LIN {X 0,Y 362.665,Z 342.074,A -85,B 0,C 180,E1 -13518.879,E2 -13518.879} C_VEL
LIN {X 0,Y 362.673,Z 345.002,A -85,B 0,C 180,E1 -13519.116,E2 -13519.116} C_VEL
LIN {X 0,Y 361.547,Z 357.376,A -85,B 0,C 180,E1 -13520.184,E2 -13520.184} C_VEL
LIN {X 0,Y 360.334,Z 368.054,A -85,B 0,C 180,E1 -13521.361,E2 -13521.361} C_VEL
LIN {X 0,Y 359.164,Z 377.919,A -85,B 0,C 180,E1 -13522.714,E2 -13522.714} C_VEL
LIN {X 0,Y 357.885,Z 387.519,A -85,B 0,C 180,E1 -13524.355,E2 -13524.355} C_VEL
LIN {X 0,Y 356.833,Z 395.168,A -85,B 0,C 180,E1 -13525.991,E2 -13525.991} C_VEL
LIN {X 0,Y 355.858,Z 401.859,A -85,B 0,C 180,E1 -13527.774,E2 -13527.774} C_VEL
LIN {X 0,Y 355.058,Z 407.359,A -85,B 0,C 180,E1 -13529.66,E2 -13529.66} C_VEL
LIN {X 0,Y 354.484,Z 411.392,A -85,B 0,C 180,E1 -13531.512,E2 -13531.512} C_VEL
LIN {X 0,Y 353.919,Z 414.746,A -85,B 0,C 180,E1 -13533.78,E2 -13533.78} C_VEL
LIN {X 0,Y 353.636,Z 416.133,A -85,B 0,C 180,E1 -13535.43,E2 -13535.43} C_VEL
LIN {X 0,Y 353.498,Z 416.697,A -85,B 0,C 180,E1 -13537.32,E2 -13537.32} C_VEL
LIN {X 0,Y 353.475,Z 415.987,A -85,B 0,C 180,E1 -13539.512,E2 -13539.512} C_VEL
LIN {X 0,Y 353.681,Z 413.711,A -85,B 0,C 180,E1 -13541.734,E2 -13541.734} C_VEL
LIN {X 0,Y 353.978,Z 411.14,A -85,B 0,C 180,E1 -13543.308,E2 -13543.308} C_VEL
LIN {X 0,Y 354.296,Z 407.587,A -85,B 0,C 180,E1 -13544.933,E2 -13544.933} C_VEL
LIN {X 0,Y 354.697,Z 403.044,A -85,B 0,C 180,E1 -13546.551,E2 -13546.551} C_VEL
LIN {X 0,Y 355.307,Z 396.31,A -85,B 0,C 180,E1 -13548.437,E2 -13548.437} C_VEL
LIN {X 0,Y 356.124,Z 388.706,A -85,B 0,C 180,E1 -13550.13,E2 -13550.13} C_VEL
LIN {X 0,Y 356.981,Z 379.715,A -85,B 0,C 180,E1 -13551.739,E2 -13551.739} C_VEL
LIN {X 0,Y 357.963,Z 369.677,A -85,B 0,C 180,E1 -13553.19,E2 -13553.19} C_VEL
LIN {X 0,Y 358.986,Z 358.544,A -85,B 0,C 180,E1 -13554.481,E2 -13554.481} C_VEL
LIN {X 0,Y 359.748,Z 347.631,A -85,B 0,C 180,E1 -13555.49,E2 -13555.49} C_VEL
LIN {X 0,Y 360.26,Z 338.398,A -85,B 0,C 180,E1 -13556.184,E2 -13556.184} C_VEL
LIN {X 0,Y 357.076,Z 324.773,A -85,B 0,C 180,E1 -13557.147,E2 -13557.147} C_VEL
LIN {X 0,Y 353.922,Z 312.67,A -85,B 0,C 180,E1 -13557.831,E2 -13557.831} C_VEL
LIN {X 0,Y 353.979,Z 310.393,A -85,B 0,C 180,E1 -13560.24,E2 -13560.24} C_VEL
LIN {X 0,Y 354.41,Z 310.341,A -85,B 0,C 180,E1 -13563.171,E2 -13563.171} C_VEL
LIN {X 0,Y 354.706,Z 310.3,A -85,B 0,C 180,E1 -13566.654,E2 -13566.654} C_VEL
LIN {X 0,Y 354.82,Z 310.289,A -85,B 0,C 180,E1 -13569.113,E2 -13569.113} C_VEL
LIN {X 0,Y 354.881,Z 310.28,A -85,B 0,C 180,E1 -13572.719,E2 -13572.719} C_VEL
LIN {X 0,Y 354.952,Z 310.269,A -85,B 0,C 180,E1 -13576.255,E2 -13576.255} C_VEL
LIN {X 0,Y 354.979,Z 310.265,A -85,B 0,C 180,E1 -13579.736,E2 -13579.736} C_VEL
LIN {X 0,Y 355.101,Z 310.253,A -85,B 0,C 180,E1 -13583.18,E2 -13583.18} C_VEL
LIN {X 0,Y 355.244,Z 310.232,A -85,B 0,C 180,E1 -13587.732,E2 -13587.732} C_VEL
LIN {X 0,Y 355.397,Z 310.213,A -85,B 0,C 180,E1 -13590,E2 -13590} C_VEL
LIN {X 0,Y 355.247,Z 310.234,A -85,B 0,C 180,E1 -13592.268,E2 -13592.268} C_VEL
LIN {X 0,Y 355.1,Z 310.254,A -85,B 0,C 180,E1 -13596.82,E2 -13596.82} C_VEL
LIN {X 0,Y 354.978,Z 310.268,A -85,B 0,C 180,E1 -13600.264,E2 -13600.264} C_VEL
LIN {X 0,Y 354.944,Z 310.271,A -85,B 0,C 180,E1 -13604.019,E2 -13604.019} C_VEL
LIN {X 0,Y 354.923,Z 310.275,A -85,B 0,C 180,E1 -13608.109,E2 -13608.109} C_VEL
LIN {X 0,Y 354.836,Z 310.287,A -85,B 0,C 180,E1 -13612.106,E2 -13612.106} C_VEL
LIN {X 0,Y 354.901,Z 310.277,A -85,B 0,C 180,E1 -13615.828,E2 -13615.828} C_VEL
LIN {X 0,Y 354.855,Z 310.282,A -85,B 0,C 180,E1 -13619.679,E2 -13619.679} C_VEL
LIN {X 0,Y 354.807,Z 310.289,A -85,B 0,C 180,E1 -13623.702,E2 -13623.702} C_VEL
LIN {X 0,Y 354.791,Z 310.289,A -85,B 0,C 180,E1 -13627.248,E2 -13627.248} C_VEL
LIN {X 0,Y 354.789,Z 310.289,A -85,B 0,C 180,E1 -13630.821,E2 -13630.821} C_VEL
LIN {X 0,Y 354.786,Z 310.289,A -85,B 0,C 180,E1 -13632.165,E2 -13632.165} C_VEL
LIN {X 0,Y 354.153,Z 310.373,A -85,B 0,C 180,E1 -13633.111,E2 -13633.111} C_VEL
LIN {X 0,Y 351.293,Z 310.729,A -85,B 0,C 180,E1 -13634.651,E2 -13634.651} C_VEL
LIN {X 0,Y 348.847,Z 311.034,A -85,B 0,C 180,E1 -13635.896,E2 -13635.896} C_VEL
LIN {X 0,Y 347.794,Z 311.16,A -85,B 0,C 180,E1 -13636.861,E2 -13636.861} C_VEL
LIN {X 0,Y 347.709,Z 311.168,A -85,B 0,C 180,E1 -13637.187,E2 -13637.187} C_VEL
LIN {X 0,Y 347.749,Z 311.167,A -85,B 0,C 180,E1 -13640.173,E2 -13640.173} C_VEL
LIN {X 0,Y 347.764,Z 311.163,A -85,B 0,C 180,E1 -13642.68,E2 -13642.68} C_VEL
LIN {X 0,Y 347.75,Z 311.168,A -85,B 0,C 180,E1 -13645.956,E2 -13645.956} C_VEL
LIN {X 0,Y 347.766,Z 311.168,A -85,B 0,C 180,E1 -13649.654,E2 -13649.654} C_VEL
LIN {X 0,Y 347.854,Z 311.153,A -85,B 0,C 180,E1 -13652.745,E2 -13652.745} C_VEL
LIN {X 0,Y 347.788,Z 311.161,A -85,B 0,C 180,E1 -13656.162,E2 -13656.162} C_VEL
LIN {X 0,Y 347.803,Z 311.16,A -85,B 0,C 180,E1 -13659.909,E2 -13659.909} C_VEL
LIN {X 0,Y 347.836,Z 311.157,A -85,B 0,C 180,E1 -13663.569,E2 -13663.569} C_VEL
LIN {X 0,Y 347.894,Z 311.152,A -85,B 0,C 180,E1 -13667.161,E2 -13667.161} C_VEL
LIN {X 0,Y 347.939,Z 311.144,A -85,B 0,C 180,E1 -13670.701,E2 -13670.701} C_VEL
LIN {X 0,Y 348.086,Z 311.129,A -85,B 0,C 180,E1 -13673.042,E2 -13673.042} C_VEL
LIN {X 0,Y 348.207,Z 311.108,A -85,B 0,C 180,E1 -13677.687,E2 -13677.687} C_VEL
LIN {X 0,Y 348.328,Z 311.093,A -85,B 0,C 180,E1 -13680,E2 -13680} C_VEL
LIN {X 0,Y 348.199,Z 311.11,A -85,B 0,C 180,E1 -13682.314,E2 -13682.314} C_VEL
LIN {X 0,Y 348.072,Z 311.129,A -85,B 0,C 180,E1 -13686.958,E2 -13686.958} C_VEL
LIN {X 0,Y 347.901,Z 311.15,A -85,B 0,C 180,E1 -13690.475,E2 -13690.475} C_VEL
LIN {X 0,Y 347.902,Z 311.148,A -85,B 0,C 180,E1 -13694.15,E2 -13694.15} C_VEL
LIN {X 0,Y 347.832,Z 311.158,A -85,B 0,C 180,E1 -13698.259,E2 -13698.259} C_VEL
LIN {X 0,Y 347.771,Z 311.163,A -85,B 0,C 180,E1 -13701.626,E2 -13701.626} C_VEL
LIN {X 0,Y 347.796,Z 311.16,A -85,B 0,C 180,E1 -13705.11,E2 -13705.11} C_VEL
LIN {X 0,Y 347.76,Z 311.164,A -85,B 0,C 180,E1 -13709.014,E2 -13709.014} C_VEL
LIN {X 0,Y 347.745,Z 311.166,A -85,B 0,C 180,E1 -13713.071,E2 -13713.071} C_VEL
LIN {X 0,Y 347.773,Z 311.167,A -85,B 0,C 180,E1 -13716.065,E2 -13716.065} C_VEL
LIN {X 0,Y 347.755,Z 311.165,A -85,B 0,C 180,E1 -13718.793,E2 -13718.793} C_VEL
LIN {X 0,Y 347.753,Z 311.169,A -85,B 0,C 180,E1 -13721.83,E2 -13721.83} C_VEL
LIN {X 0,Y 347.791,Z 311.271,A -85,B 0,C 180,E1 -13724.819,E2 -13724.819} C_VEL
LIN {X 0,Y 348.908,Z 317.424,A -85,B 0,C 180,E1 -13728.339,E2 -13728.339} C_VEL
LIN {X 0,Y 349.989,Z 323.328,A -85,B 0,C 180,E1 -13731.55,E2 -13731.55} C_VEL
LIN {X 0,Y 350.336,Z 327.895,A -85,B 0,C 180,E1 -13733.897,E2 -13733.897} C_VEL
LIN {X 0,Y 349.502,Z 334.535,A -85,B 0,C 180,E1 -13737.116,E2 -13737.116} C_VEL
LIN {X 0,Y 348.554,Z 342.889,A -85,B 0,C 180,E1 -13741.058,E2 -13741.058} C_VEL
LIN {X 0,Y 347.745,Z 351.233,A -85,B 0,C 180,E1 -13744.886,E2 -13744.886} C_VEL
LIN {X 0,Y 347.106,Z 359.56,A -85,B 0,C 180,E1 -13748.652,E2 -13748.652} C_VEL
LIN {X 0,Y 346.983,Z 362.085,A -85,B 0,C 180,E1 -13749.782,E2 -13749.782} C_VEL
LIN {X 0,Y 348.977,Z 376.53,A -85,B 0,C 180,E1 -13750.44,E2 -13750.44} C_VEL
LIN {X 0,Y 350.363,Z 388.913,A -85,B 0,C 180,E1 -13751.22,E2 -13751.22} C_VEL
LIN {X 0,Y 351.311,Z 401.597,A -85,B 0,C 180,E1 -13752.237,E2 -13752.237} C_VEL
LIN {X 0,Y 351.019,Z 407.958,A -85,B 0,C 180,E1 -13752.823,E2 -13752.823} C_VEL
LIN {X 0,Y 349.791,Z 419.655,A -85,B 0,C 180,E1 -13754.112,E2 -13754.112} C_VEL
LIN {X 0,Y 348.824,Z 429.132,A -85,B 0,C 180,E1 -13755.41,E2 -13755.41} C_VEL
LIN {X 0,Y 348.012,Z 437.864,A -85,B 0,C 180,E1 -13756.868,E2 -13756.868} C_VEL
LIN {X 0,Y 347.235,Z 446.325,A -85,B 0,C 180,E1 -13758.619,E2 -13758.619} C_VEL
LIN {X 0,Y 346.77,Z 453.136,A -85,B 0,C 180,E1 -13760.375,E2 -13760.375} C_VEL
LIN {X 0,Y 346.461,Z 459.371,A -85,B 0,C 180,E1 -13762.423,E2 -13762.423} C_VEL
LIN {X 0,Y 346.36,Z 463.393,A -85,B 0,C 180,E1 -13764.177,E2 -13764.177} C_VEL
LIN {X 0,Y 346.372,Z 465.449,A -85,B 0,C 180,E1 -13765.345,E2 -13765.345} C_VEL
LIN {X 0,Y 346.529,Z 468.273,A -85,B 0,C 180,E1 -13767.675,E2 -13767.675} C_VEL
LIN {X 0,Y 346.531,Z 469.026,A -85,B 0,C 180,E1 -13768.838,E2 -13768.838} C_VEL
LIN {X 0,Y 346.546,Z 469.344,A -85,B 0,C 180,E1 -13770,E2 -13770} C_VEL
LIN {X 0,Y 346.51,Z 469.256,A -85,B 0,C 180,E1 -13771.162,E2 -13771.162} C_VEL
LIN {X 0,Y 346.497,Z 468.769,A -85,B 0,C 180,E1 -13772.325,E2 -13772.325} C_VEL
LIN {X 0,Y 346.337,Z 467.838,A -85,B 0,C 180,E1 -13773.49,E2 -13773.49} C_VEL
LIN {X 0,Y 346.321,Z 466.48,A -85,B 0,C 180,E1 -13774.656,E2 -13774.656} C_VEL
LIN {X 0,Y 346.243,Z 464.483,A -85,B 0,C 180,E1 -13775.956,E2 -13775.956} C_VEL
LIN {X 0,Y 346.409,Z 461.197,A -85,B 0,C 180,E1 -13777.578,E2 -13777.578} C_VEL
LIN {X 0,Y 346.684,Z 456.619,A -85,B 0,C 180,E1 -13779.333,E2 -13779.333} C_VEL
LIN {X 0,Y 347.291,Z 449.778,A -85,B 0,C 180,E1 -13781.38,E2 -13781.38} C_VEL
LIN {X 0,Y 348.248,Z 442.357,A -85,B 0,C 180,E1 -13783.123,E2 -13783.123} C_VEL
LIN {X 0,Y 349.358,Z 433.079,A -85,B 0,C 180,E1 -13784.888,E2 -13784.888} C_VEL
LIN {X 0,Y 350.468,Z 423.926,A -85,B 0,C 180,E1 -13786.305,E2 -13786.305} C_VEL
LIN {X 0,Y 352.052,Z 412.428,A -85,B 0,C 180,E1 -13787.724,E2 -13787.724} C_VEL
LIN {X 0,Y 352.831,Z 404.137,A -85,B 0,C 180,E1 -13788.585,E2 -13788.585} C_VEL
LIN {X 0,Y 352.469,Z 391.587,A -85,B 0,C 180,E1 -13789.73,E2 -13789.73} C_VEL
LIN {X 0,Y 351.594,Z 381.993,A -85,B 0,C 180,E1 -13790.475,E2 -13790.475} C_VEL
LIN {X 0,Y 349.591,Z 369.477,A -85,B 0,C 180,E1 -13791.313,E2 -13791.313} C_VEL
LIN {X 0,Y 347.227,Z 358.557,A -85,B 0,C 180,E1 -13791.943,E2 -13791.943} C_VEL
LIN {X 0,Y 347.858,Z 350.269,A -85,B 0,C 180,E1 -13795.746,E2 -13795.746} C_VEL
LIN {X 0,Y 348.678,Z 342.519,A -85,B 0,C 180,E1 -13799.442,E2 -13799.442} C_VEL
LIN {X 0,Y 349.811,Z 334.351,A -85,B 0,C 180,E1 -13803.539,E2 -13803.539} C_VEL
LIN {X 0,Y 350.574,Z 329.466,A -85,B 0,C 180,E1 -13806.13,E2 -13806.13} C_VEL
LIN {X 0,Y 350.555,Z 326.753,A -85,B 0,C 180,E1 -13807.696,E2 -13807.696} C_VEL
LIN {X 0,Y 349.769,Z 321.77,A -85,B 0,C 180,E1 -13810.835,E2 -13810.835} C_VEL
LIN {X 0,Y 349.048,Z 317.863,A -85,B 0,C 180,E1 -13813.543,E2 -13813.543} C_VEL
LIN {X 0,Y 348.264,Z 313.827,A -85,B 0,C 180,E1 -13816.676,E2 -13816.676} C_VEL
LIN {X 0,Y 347.745,Z 311.176,A -85,B 0,C 180,E1 -13819.035,E2 -13819.035} C_VEL
LIN {X 0,Y 347.769,Z 311.169,A -85,B 0,C 180,E1 -13822.68,E2 -13822.68} C_VEL
LIN {X 0,Y 347.752,Z 311.169,A -85,B 0,C 180,E1 -13825.956,E2 -13825.956} C_VEL
LIN {X 0,Y 347.768,Z 311.167,A -85,B 0,C 180,E1 -13829.654,E2 -13829.654} C_VEL
LIN {X 0,Y 347.856,Z 311.156,A -85,B 0,C 180,E1 -13832.745,E2 -13832.745} C_VEL
LIN {X 0,Y 347.793,Z 311.162,A -85,B 0,C 180,E1 -13836.162,E2 -13836.162} C_VEL
LIN {X 0,Y 347.822,Z 311.157,A -85,B 0,C 180,E1 -13839.91,E2 -13839.91} C_VEL
LIN {X 0,Y 347.871,Z 311.151,A -85,B 0,C 180,E1 -13842.359,E2 -13842.359} C_VEL
LIN {X 0,Y 347.901,Z 311.15,A -85,B 0,C 180,E1 -13845.971,E2 -13845.971} C_VEL
LIN {X 0,Y 347.901,Z 311.149,A -85,B 0,C 180,E1 -13849.525,E2 -13849.525} C_VEL
LIN {X 0,Y 348.072,Z 311.127,A -85,B 0,C 180,E1 -13853.042,E2 -13853.042} C_VEL
LIN {X 0,Y 348.21,Z 311.111,A -85,B 0,C 180,E1 -13857.686,E2 -13857.686} C_VEL
LIN {X 0,Y 348.35,Z 311.096,A -85,B 0,C 180,E1 -13860,E2 -13860} C_VEL
LIN {X 0,Y 348.213,Z 311.111,A -85,B 0,C 180,E1 -13862.313,E2 -13862.313} C_VEL
LIN {X 0,Y 348.069,Z 311.13,A -85,B 0,C 180,E1 -13866.958,E2 -13866.958} C_VEL
LIN {X 0,Y 347.992,Z 311.14,A -85,B 0,C 180,E1 -13868.268,E2 -13868.268} C_VEL
LIN {X 0,Y 347.82,Z 313.428,A -85,B 0,C 180,E1 -13871.657,E2 -13871.657} C_VEL
LIN {X 0,Y 347.641,Z 316.115,A -85,B 0,C 180,E1 -13875.237,E2 -13875.237} C_VEL
LIN {X 0,Y 347.621,Z 317.069,A -85,B 0,C 180,E1 -13876.253,E2 -13876.253} C_VEL
LIN {X 0,Y 352.283,Z 329.9,A -85,B 0,C 180,E1 -13877.263,E2 -13877.263} C_VEL
LIN {X 0,Y 355.595,Z 341.553,A -85,B 0,C 180,E1 -13878.3,E2 -13878.3} C_VEL
LIN {X 0,Y 356.194,Z 344.142,A -85,B 0,C 180,E1 -13878.551,E2 -13878.551} C_VEL
LIN {X 0,Y 355.247,Z 355.316,A -85,B 0,C 180,E1 -13879.502,E2 -13879.502} C_VEL
LIN {X 0,Y 354.027,Z 365.973,A -85,B 0,C 180,E1 -13880.632,E2 -13880.632} C_VEL
LIN {X 0,Y 352.857,Z 375.772,A -85,B 0,C 180,E1 -13881.929,E2 -13881.929} C_VEL
LIN {X 0,Y 351.41,Z 385.788,A -85,B 0,C 180,E1 -13883.577,E2 -13883.577} C_VEL
LIN {X 0,Y 350.332,Z 393.517,A -85,B 0,C 180,E1 -13885.156,E2 -13885.156} C_VEL
LIN {X 0,Y 349.251,Z 400.486,A -85,B 0,C 180,E1 -13886.918,E2 -13886.918} C_VEL
LIN {X 0,Y 348.303,Z 406.735,A -85,B 0,C 180,E1 -13888.964,E2 -13888.964} C_VEL
LIN {X 0,Y 347.584,Z 411.468,A -85,B 0,C 180,E1 -13891.037,E2 -13891.037} C_VEL
LIN {X 0,Y 346.981,Z 414.757,A -85,B 0,C 180,E1 -13893.153,E2 -13893.153} C_VEL
LIN {X 0,Y 346.698,Z 416.206,A -85,B 0,C 180,E1 -13894.583,E2 -13894.583} C_VEL
LIN {X 0,Y 346.501,Z 417.022,A -85,B 0,C 180,E1 -13896.029,E2 -13896.029} C_VEL
LIN {X 0,Y 346.402,Z 417.224,A -85,B 0,C 180,E1 -13897.696,E2 -13897.696} C_VEL
LIN {X 0,Y 346.395,Z 416.473,A -85,B 0,C 180,E1 -13899.557,E2 -13899.557} C_VEL
LIN {X 0,Y 346.554,Z 414.734,A -85,B 0,C 180,E1 -13901.379,E2 -13901.379} C_VEL
LIN {X 0,Y 346.943,Z 411.334,A -85,B 0,C 180,E1 -13903.53,E2 -13903.53} C_VEL
LIN {X 0,Y 347.269,Z 407.89,A -85,B 0,C 180,E1 -13905.099,E2 -13905.099} C_VEL
LIN {X 0,Y 347.789,Z 402.248,A -85,B 0,C 180,E1 -13907.075,E2 -13907.075} C_VEL
LIN {X 0,Y 348.349,Z 396.36,A -85,B 0,C 180,E1 -13908.702,E2 -13908.702} C_VEL
LIN {X 0,Y 349.146,Z 389.139,A -85,B 0,C 180,E1 -13910.326,E2 -13910.326} C_VEL
LIN {X 0,Y 350.002,Z 380.39,A -85,B 0,C 180,E1 -13911.923,E2 -13911.923} C_VEL
LIN {X 0,Y 350.969,Z 370.922,A -85,B 0,C 180,E1 -13913.329,E2 -13913.329} C_VEL
LIN {X 0,Y 351.978,Z 360.255,A -85,B 0,C 180,E1 -13914.616,E2 -13914.616} C_VEL
LIN {X 0,Y 352.791,Z 349.433,A -85,B 0,C 180,E1 -13915.666,E2 -13915.666} C_VEL
LIN {X 0,Y 353.507,Z 340.69,A -85,B 0,C 180,E1 -13916.346,E2 -13916.346} C_VEL
LIN {X 0,Y 350.753,Z 328.113,A -85,B 0,C 180,E1 -13917.291,E2 -13917.291} C_VEL
LIN {X 0,Y 347.373,Z 315.098,A -85,B 0,C 180,E1 -13918.049,E2 -13918.049} C_VEL
LIN {X 0,Y 346.908,Z 313.147,A -85,B 0,C 180,E1 -13918.172,E2 -13918.172} C_VEL
LIN {X 0,Y 346.898,Z 311.778,A -85,B 0,C 180,E1 -13919.569,E2 -13919.569} C_VEL
LIN {X 0,Y 347.058,Z 311.255,A -85,B 0,C 180,E1 -13920.921,E2 -13920.921} C_VEL
LIN {X 0,Y 347.381,Z 311.215,A -85,B 0,C 180,E1 -13923.571,E2 -13923.571} C_VEL
LIN {X 0,Y 347.632,Z 311.18,A -85,B 0,C 180,E1 -13926.15,E2 -13926.15} C_VEL
LIN {X 0,Y 347.796,Z 311.16,A -85,B 0,C 180,E1 -13929.908,E2 -13929.908} C_VEL
LIN {X 0,Y 347.833,Z 311.156,A -85,B 0,C 180,E1 -13933.568,E2 -13933.568} C_VEL
LIN {X 0,Y 347.891,Z 311.152,A -85,B 0,C 180,E1 -13937.16,E2 -13937.16} C_VEL
LIN {X 0,Y 347.942,Z 311.145,A -85,B 0,C 180,E1 -13940.701,E2 -13940.701} C_VEL
LIN {X 0,Y 348.051,Z 311.128,A -85,B 0,C 180,E1 -13944.205,E2 -13944.205} C_VEL
LIN {X 0,Y 348.207,Z 311.108,A -85,B 0,C 180,E1 -13947.686,E2 -13947.686} C_VEL
LIN {X 0,Y 348.346,Z 311.091,A -85,B 0,C 180,E1 -13950,E2 -13950} C_VEL
LIN {X 0,Y 348.209,Z 311.11,A -85,B 0,C 180,E1 -13952.313,E2 -13952.313} C_VEL
LIN {X 0,Y 348.068,Z 311.128,A -85,B 0,C 180,E1 -13956.958,E2 -13956.958} C_VEL
LIN {X 0,Y 347.929,Z 311.148,A -85,B 0,C 180,E1 -13960.474,E2 -13960.474} C_VEL
LIN {X 0,Y 347.899,Z 311.15,A -85,B 0,C 180,E1 -13964.15,E2 -13964.15} C_VEL
LIN {X 0,Y 347.892,Z 311.153,A -85,B 0,C 180,E1 -13968.29,E2 -13968.29} C_VEL
LIN {X 0,Y 347.79,Z 311.161,A -85,B 0,C 180,E1 -13971.635,E2 -13971.635} C_VEL
LIN {X 0,Y 347.813,Z 311.157,A -85,B 0,C 180,E1 -13975.109,E2 -13975.109} C_VEL
LIN {X 0,Y 347.812,Z 311.159,A -85,B 0,C 180,E1 -13977.694,E2 -13977.694} C_VEL
LIN {X 0,Y 347.765,Z 311.167,A -85,B 0,C 180,E1 -13980.347,E2 -13980.347} C_VEL
LIN {X 0,Y 347.745,Z 311.168,A -85,B 0,C 180,E1 -13984.464,E2 -13984.464} C_VEL
LIN {X 0,Y 347.775,Z 311.167,A -85,B 0,C 180,E1 -13987.989,E2 -13987.989} C_VEL
LIN {X 0,Y 347.752,Z 311.17,A -85,B 0,C 180,E1 -13991.83,E2 -13991.83} C_VEL
LIN {X 0,Y 347.707,Z 311.171,A -85,B 0,C 180,E1 -13995.027,E2 -13995.027} C_VEL
LIN {X 0,Y 347.709,Z 311.168,A -85,B 0,C 180,E1 -13997.187,E2 -13997.187} C_VEL
LIN {X 0,Y 347.053,Z 311.255,A -85,B 0,C 180,E1 -13998.154,E2 -13998.154} C_VEL
LIN {X 0,Y 344.233,Z 311.608,A -85,B 0,C 180,E1 -13999.728,E2 -13999.728} C_VEL
LIN {X 0,Y 341.834,Z 311.907,A -85,B 0,C 180,E1 -14001.001,E2 -14001.001} C_VEL
LIN {X 0,Y 340.79,Z 312.035,A -85,B 0,C 180,E1 -14001.986,E2 -14001.986} C_VEL
LIN {X 0,Y 340.698,Z 312.044,A -85,B 0,C 180,E1 -14002.32,E2 -14002.32} C_VEL
LIN {X 0,Y 340.725,Z 312.046,A -85,B 0,C 180,E1 -14005.596,E2 -14005.596} C_VEL
LIN {X 0,Y 340.706,Z 312.044,A -85,B 0,C 180,E1 -14008.956,E2 -14008.956} C_VEL
LIN {X 0,Y 340.781,Z 312.033,A -85,B 0,C 180,E1 -14012.474,E2 -14012.474} C_VEL
LIN {X 0,Y 340.757,Z 312.04,A -85,B 0,C 180,E1 -14015.639,E2 -14015.639} C_VEL
LIN {X 0,Y 340.733,Z 312.043,A -85,B 0,C 180,E1 -14019.473,E2 -14019.473} C_VEL
LIN {X 0,Y 340.795,Z 312.032,A -85,B 0,C 180,E1 -14021.981,E2 -14021.981} C_VEL
LIN {X 0,Y 340.873,Z 312.023,A -85,B 0,C 180,E1 -14025.705,E2 -14025.705} C_VEL
LIN {X 0,Y 340.852,Z 312.028,A -85,B 0,C 180,E1 -14029.306,E2 -14029.306} C_VEL
LIN {X 0,Y 341.053,Z 312.004,A -85,B 0,C 180,E1 -14032.898,E2 -14032.898} C_VEL
LIN {X 0,Y 341.169,Z 311.985,A -85,B 0,C 180,E1 -14037.639,E2 -14037.639} C_VEL
LIN {X 0,Y 341.279,Z 311.971,A -85,B 0,C 180,E1 -14040,E2 -14040} C_VEL
LIN {X 0,Y 341.16,Z 311.987,A -85,B 0,C 180,E1 -14042.361,E2 -14042.361} C_VEL
LIN {X 0,Y 341.02,Z 312.006,A -85,B 0,C 180,E1 -14047.103,E2 -14047.103} C_VEL
LIN {X 0,Y 340.853,Z 312.029,A -85,B 0,C 180,E1 -14050.695,E2 -14050.695} C_VEL
LIN {X 0,Y 340.867,Z 312.026,A -85,B 0,C 180,E1 -14054.325,E2 -14054.325} C_VEL
LIN {X 0,Y 340.789,Z 312.037,A -85,B 0,C 180,E1 -14058.44,E2 -14058.44} C_VEL
LIN {X 0,Y 340.721,Z 312.041,A -85,B 0,C 180,E1 -14061.842,E2 -14061.842} C_VEL
LIN {X 0,Y 340.748,Z 312.038,A -85,B 0,C 180,E1 -14065.667,E2 -14065.667} C_VEL
LIN {X 0,Y 340.735,Z 312.04,A -85,B 0,C 180,E1 -14069.672,E2 -14069.672} C_VEL
LIN {X 0,Y 340.697,Z 312.046,A -85,B 0,C 180,E1 -14073.846,E2 -14073.846} C_VEL
LIN {X 0,Y 340.708,Z 312.043,A -85,B 0,C 180,E1 -14076.742,E2 -14076.742} C_VEL
LIN {X 0,Y 340.691,Z 312.049,A -85,B 0,C 180,E1 -14080.247,E2 -14080.247} C_VEL
LIN {X 0,Y 340.676,Z 312.05,A -85,B 0,C 180,E1 -14083.777,E2 -14083.777} C_VEL
LIN {X 0,Y 340.745,Z 312.183,A -85,B 0,C 180,E1 -14084.529,E2 -14084.529} C_VEL
LIN {X 0,Y 341.943,Z 318.683,A -85,B 0,C 180,E1 -14088.333,E2 -14088.333} C_VEL
LIN {X 0,Y 343.148,Z 325.501,A -85,B 0,C 180,E1 -14092.089,E2 -14092.089} C_VEL
LIN {X 0,Y 343.319,Z 328.345,A -85,B 0,C 180,E1 -14093.583,E2 -14093.583} C_VEL
LIN {X 0,Y 342.676,Z 333.956,A -85,B 0,C 180,E1 -14096.375,E2 -14096.375} C_VEL
LIN {X 0,Y 341.648,Z 342.287,A -85,B 0,C 180,E1 -14100.416,E2 -14100.416} C_VEL
LIN {X 0,Y 340.757,Z 350.593,A -85,B 0,C 180,E1 -14104.334,E2 -14104.334} C_VEL
LIN {X 0,Y 340.066,Z 359.448,A -85,B 0,C 180,E1 -14108.435,E2 -14108.435} C_VEL
LIN {X 0,Y 339.928,Z 361.604,A -85,B 0,C 180,E1 -14109.422,E2 -14109.422} C_VEL
LIN {X 0,Y 341.965,Z 376.241,A -85,B 0,C 180,E1 -14110.111,E2 -14110.111} C_VEL
LIN {X 0,Y 343.395,Z 389.241,A -85,B 0,C 180,E1 -14110.958,E2 -14110.958} C_VEL
LIN {X 0,Y 344.251,Z 400.211,A -85,B 0,C 180,E1 -14111.86,E2 -14111.86} C_VEL
LIN {X 0,Y 344.242,Z 406.734,A -85,B 0,C 180,E1 -14112.474,E2 -14112.474} C_VEL
LIN {X 0,Y 343.04,Z 417.408,A -85,B 0,C 180,E1 -14113.638,E2 -14113.638} C_VEL
LIN {X 0,Y 342.012,Z 427.255,A -85,B 0,C 180,E1 -14114.974,E2 -14114.974} C_VEL
LIN {X 0,Y 341.265,Z 435.32,A -85,B 0,C 180,E1 -14116.3,E2 -14116.3} C_VEL
LIN {X 0,Y 340.41,Z 444.216,A -85,B 0,C 180,E1 -14118.085,E2 -14118.085} C_VEL
LIN {X 0,Y 339.777,Z 451.344,A -85,B 0,C 180,E1 -14119.874,E2 -14119.874} C_VEL
LIN {X 0,Y 339.453,Z 457.025,A -85,B 0,C 180,E1 -14121.667,E2 -14121.667} C_VEL
LIN {X 0,Y 339.338,Z 462.166,A -85,B 0,C 180,E1 -14123.788,E2 -14123.788} C_VEL
LIN {X 0,Y 339.305,Z 464.811,A -85,B 0,C 180,E1 -14125.247,E2 -14125.247} C_VEL
LIN {X 0,Y 339.28,Z 466.443,A -85,B 0,C 180,E1 -14126.437,E2 -14126.437} C_VEL
LIN {X 0,Y 339.462,Z 467.672,A -85,B 0,C 180,E1 -14127.627,E2 -14127.627} C_VEL
LIN {X 0,Y 339.465,Z 468.458,A -85,B 0,C 180,E1 -14128.814,E2 -14128.814} C_VEL
LIN {X 0,Y 339.476,Z 468.792,A -85,B 0,C 180,E1 -14130,E2 -14130} C_VEL
LIN {X 0,Y 339.445,Z 468.719,A -85,B 0,C 180,E1 -14131.186,E2 -14131.186} C_VEL
LIN {X 0,Y 339.413,Z 468.246,A -85,B 0,C 180,E1 -14132.373,E2 -14132.373} C_VEL
LIN {X 0,Y 339.251,Z 467.349,A -85,B 0,C 180,E1 -14133.563,E2 -14133.563} C_VEL
LIN {X 0,Y 339.226,Z 466.01,A -85,B 0,C 180,E1 -14134.754,E2 -14134.754} C_VEL
LIN {X 0,Y 339.227,Z 463.224,A -85,B 0,C 180,E1 -14136.543,E2 -14136.543} C_VEL
LIN {X 0,Y 339.419,Z 459.417,A -85,B 0,C 180,E1 -14138.334,E2 -14138.334} C_VEL
LIN {X 0,Y 339.781,Z 454.495,A -85,B 0,C 180,E1 -14140.126,E2 -14140.126} C_VEL
LIN {X 0,Y 340.621,Z 447.176,A -85,B 0,C 180,E1 -14142.21,E2 -14142.21} C_VEL
LIN {X 0,Y 341.584,Z 439.32,A -85,B 0,C 180,E1 -14143.99,E2 -14143.99} C_VEL
LIN {X 0,Y 342.628,Z 431.371,A -85,B 0,C 180,E1 -14145.466,E2 -14145.466} C_VEL
LIN {X 0,Y 344.099,Z 420.723,A -85,B 0,C 180,E1 -14147.074,E2 -14147.074} C_VEL
LIN {X 0,Y 345.625,Z 410.03,A -85,B 0,C 180,E1 -14148.372,E2 -14148.372} C_VEL
LIN {X 0,Y 346.063,Z 403.049,A -85,B 0,C 180,E1 -14149.105,E2 -14149.105} C_VEL
LIN {X 0,Y 345.732,Z 391.118,A -85,B 0,C 180,E1 -14150.217,E2 -14150.217} C_VEL
LIN {X 0,Y 344.502,Z 379.491,A -85,B 0,C 180,E1 -14151.143,E2 -14151.143} C_VEL
LIN {X 0,Y 342.3,Z 366.872,A -85,B 0,C 180,E1 -14152.007,E2 -14152.007} C_VEL
LIN {X 0,Y 340.246,Z 357.904,A -85,B 0,C 180,E1 -14152.553,E2 -14152.553} C_VEL
LIN {X 0,Y 340.918,Z 349.948,A -85,B 0,C 180,E1 -14156.31,E2 -14156.31} C_VEL
LIN {X 0,Y 341.66,Z 343.272,A -85,B 0,C 180,E1 -14159.583,E2 -14159.583} C_VEL
LIN {X 0,Y 342.817,Z 335.455,A -85,B 0,C 180,E1 -14163.609,E2 -14163.609} C_VEL
LIN {X 0,Y 343.614,Z 330.352,A -85,B 0,C 180,E1 -14166.381,E2 -14166.381} C_VEL
LIN {X 0,Y 343.574,Z 327.877,A -85,B 0,C 180,E1 -14167.856,E2 -14167.856} C_VEL
LIN {X 0,Y 342.794,Z 323.002,A -85,B 0,C 180,E1 -14171.001,E2 -14171.001} C_VEL
LIN {X 0,Y 341.911,Z 318.413,A -85,B 0,C 180,E1 -14174.337,E2 -14174.337} C_VEL
LIN {X 0,Y 341.101,Z 314.11,A -85,B 0,C 180,E1 -14177.88,E2 -14177.88} C_VEL
LIN {X 0,Y 340.723,Z 312.047,A -85,B 0,C 180,E1 -14180,E2 -14180} C_VEL
LIN {X 0,Y 340.715,Z 312.044,A -85,B 0,C 180,E1 -14183.559,E2 -14183.559} C_VEL
LIN {X 0,Y 340.698,Z 312.049,A -85,B 0,C 180,E1 -14186.154,E2 -14186.154} C_VEL
LIN {X 0,Y 340.778,Z 312.038,A -85,B 0,C 180,E1 -14190.333,E2 -14190.333} C_VEL
LIN {X 0,Y 340.809,Z 312.033,A -85,B 0,C 180,E1 -14193.02,E2 -14193.02} C_VEL
LIN {X 0,Y 340.733,Z 312.043,A -85,B 0,C 180,E1 -14196.927,E2 -14196.927} C_VEL
LIN {X 0,Y 340.799,Z 312.035,A -85,B 0,C 180,E1 -14200.734,E2 -14200.734} C_VEL
LIN {X 0,Y 340.791,Z 312.037,A -85,B 0,C 180,E1 -14203.219,E2 -14203.219} C_VEL
LIN {X 0,Y 340.849,Z 312.025,A -85,B 0,C 180,E1 -14206.89,E2 -14206.89} C_VEL
LIN {X 0,Y 340.886,Z 312.024,A -85,B 0,C 180,E1 -14210.506,E2 -14210.506} C_VEL
LIN {X 0,Y 341.029,Z 312.006,A -85,B 0,C 180,E1 -14214.086,E2 -14214.086} C_VEL
LIN {X 0,Y 341.172,Z 311.987,A -85,B 0,C 180,E1 -14217.639,E2 -14217.639} C_VEL
LIN {X 0,Y 341.3,Z 311.974,A -85,B 0,C 180,E1 -14220,E2 -14220} C_VEL
LIN {X 0,Y 341.174,Z 311.988,A -85,B 0,C 180,E1 -14222.361,E2 -14222.361} C_VEL
LIN {X 0,Y 341.015,Z 312.009,A -85,B 0,C 180,E1 -14227.103,E2 -14227.103} C_VEL
LIN {X 0,Y 340.967,Z 312.304,A -85,B 0,C 180,E1 -14228.356,E2 -14228.356} C_VEL
LIN {X 0,Y 340.806,Z 314.786,A -85,B 0,C 180,E1 -14231.901,E2 -14231.901} C_VEL
LIN {X 0,Y 340.621,Z 317.483,A -85,B 0,C 180,E1 -14235.559,E2 -14235.559} C_VEL
LIN {X 0,Y 340.601,Z 317.545,A -85,B 0,C 180,E1 -14235.636,E2 -14235.636} C_VEL
LIN {X 0,Y 342.771,Z 323.304,A -85,B 0,C 180,E1 -14236.091,E2 -14236.091} C_VEL
LIN {X 0,Y 346.749,Z 334.691,A -85,B 0,C 180,E1 -14237.091,E2 -14237.091} C_VEL
LIN {X 0,Y 349.601,Z 345.658,A -85,B 0,C 180,E1 -14238.155,E2 -14238.155} C_VEL
LIN {X 0,Y 348.537,Z 357.633,A -85,B 0,C 180,E1 -14239.221,E2 -14239.221} C_VEL
LIN {X 0,Y 347.262,Z 368.127,A -85,B 0,C 180,E1 -14240.397,E2 -14240.397} C_VEL
LIN {X 0,Y 345.826,Z 378.965,A -85,B 0,C 180,E1 -14241.927,E2 -14241.927} C_VEL
LIN {X 0,Y 344.561,Z 387.33,A -85,B 0,C 180,E1 -14243.383,E2 -14243.383} C_VEL
LIN {X 0,Y 343.308,Z 395.452,A -85,B 0,C 180,E1 -14245.137,E2 -14245.137} C_VEL
LIN {X 0,Y 342.26,Z 401.842,A -85,B 0,C 180,E1 -14246.856,E2 -14246.856} C_VEL
LIN {X 0,Y 341.266,Z 407.929,A -85,B 0,C 180,E1 -14248.944,E2 -14248.944} C_VEL
LIN {X 0,Y 340.524,Z 412.465,A -85,B 0,C 180,E1 -14251.062,E2 -14251.062} C_VEL
LIN {X 0,Y 340.082,Z 414.717,A -85,B 0,C 180,E1 -14252.5,E2 -14252.5} C_VEL
LIN {X 0,Y 339.706,Z 416.519,A -85,B 0,C 180,E1 -14254.153,E2 -14254.153} C_VEL
LIN {X 0,Y 339.435,Z 417.654,A -85,B 0,C 180,E1 -14256.147,E2 -14256.147} C_VEL
LIN {X 0,Y 339.31,Z 417.594,A -85,B 0,C 180,E1 -14258.417,E2 -14258.417} C_VEL
LIN {X 0,Y 339.357,Z 416.669,A -85,B 0,C 180,E1 -14259.98,E2 -14259.98} C_VEL
LIN {X 0,Y 339.54,Z 414.687,A -85,B 0,C 180,E1 -14261.828,E2 -14261.828} C_VEL
LIN {X 0,Y 339.892,Z 411.741,A -85,B 0,C 180,E1 -14263.639,E2 -14263.639} C_VEL
LIN {X 0,Y 340.344,Z 406.901,A -85,B 0,C 180,E1 -14265.78,E2 -14265.78} C_VEL
LIN {X 0,Y 340.845,Z 401.927,A -85,B 0,C 180,E1 -14267.455,E2 -14267.455} C_VEL
LIN {X 0,Y 341.466,Z 395.79,A -85,B 0,C 180,E1 -14269.124,E2 -14269.124} C_VEL
LIN {X 0,Y 342.34,Z 387.757,A -85,B 0,C 180,E1 -14270.885,E2 -14270.885} C_VEL
LIN {X 0,Y 343.346,Z 378.445,A -85,B 0,C 180,E1 -14272.537,E2 -14272.537} C_VEL
LIN {X 0,Y 344.367,Z 368.637,A -85,B 0,C 180,E1 -14273.941,E2 -14273.941} C_VEL
LIN {X 0,Y 345.379,Z 357.121,A -85,B 0,C 180,E1 -14275.266,E2 -14275.266} C_VEL
LIN {X 0,Y 346.346,Z 345.74,A -85,B 0,C 180,E1 -14276.301,E2 -14276.301} C_VEL
LIN {X 0,Y 346.537,Z 340.847,A -85,B 0,C 180,E1 -14276.68,E2 -14276.68} C_VEL
LIN {X 0,Y 343.596,Z 328.031,A -85,B 0,C 180,E1 -14277.655,E2 -14277.655} C_VEL
LIN {X 0,Y 340.145,Z 315.11,A -85,B 0,C 180,E1 -14278.423,E2 -14278.423} C_VEL
LIN {X 0,Y 339.838,Z 313.637,A -85,B 0,C 180,E1 -14278.517,E2 -14278.517} C_VEL
LIN {X 0,Y 339.905,Z 312.145,A -85,B 0,C 180,E1 -14280.274,E2 -14280.274} C_VEL
LIN {X 0,Y 340.293,Z 312.097,A -85,B 0,C 180,E1 -14282.976,E2 -14282.976} C_VEL
LIN {X 0,Y 340.555,Z 312.064,A -85,B 0,C 180,E1 -14285.623,E2 -14285.623} C_VEL
LIN {X 0,Y 340.705,Z 312.043,A -85,B 0,C 180,E1 -14288.204,E2 -14288.204} C_VEL
LIN {X 0,Y 340.793,Z 312.032,A -85,B 0,C 180,E1 -14291.981,E2 -14291.981} C_VEL
LIN {X 0,Y 340.87,Z 312.023,A -85,B 0,C 180,E1 -14295.705,E2 -14295.705} C_VEL
LIN {X 0,Y 340.872,Z 312.025,A -85,B 0,C 180,E1 -14299.306,E2 -14299.306} C_VEL
LIN {X 0,Y 341.017,Z 312.009,A -85,B 0,C 180,E1 -14302.897,E2 -14302.897} C_VEL
LIN {X 0,Y 341.168,Z 311.985,A -85,B 0,C 180,E1 -14307.639,E2 -14307.639} C_VEL
LIN {X 0,Y 341.296,Z 311.969,A -85,B 0,C 180,E1 -14310,E2 -14310} C_VEL
LIN {X 0,Y 341.171,Z 311.987,A -85,B 0,C 180,E1 -14312.361,E2 -14312.361} C_VEL
LIN {X 0,Y 341.017,Z 312.005,A -85,B 0,C 180,E1 -14317.103,E2 -14317.103} C_VEL
LIN {X 0,Y 340.871,Z 312.026,A -85,B 0,C 180,E1 -14320.694,E2 -14320.694} C_VEL
LIN {X 0,Y 340.864,Z 312.028,A -85,B 0,C 180,E1 -14324.325,E2 -14324.325} C_VEL
LIN {X 0,Y 340.838,Z 312.031,A -85,B 0,C 180,E1 -14328.467,E2 -14328.467} C_VEL
LIN {X 0,Y 340.755,Z 312.038,A -85,B 0,C 180,E1 -14331.857,E2 -14331.857} C_VEL
LIN {X 0,Y 340.774,Z 312.035,A -85,B 0,C 180,E1 -14335.664,E2 -14335.664} C_VEL
LIN {X 0,Y 340.742,Z 312.042,A -85,B 0,C 180,E1 -14338.32,E2 -14338.32} C_VEL
LIN {X 0,Y 340.705,Z 312.043,A -85,B 0,C 180,E1 -14341.044,E2 -14341.044} C_VEL
LIN {X 0,Y 340.719,Z 312.041,A -85,B 0,C 180,E1 -14345.279,E2 -14345.279} C_VEL
LIN {X 0,Y 340.711,Z 312.044,A -85,B 0,C 180,E1 -14348.386,E2 -14348.386} C_VEL
LIN {X 0,Y 340.7,Z 312.048,A -85,B 0,C 180,E1 -14352.046,E2 -14352.046} C_VEL
LIN {X 0,Y 340.654,Z 312.051,A -85,B 0,C 180,E1 -14356.227,E2 -14356.227} C_VEL
LIN {X 0,Y 340.691,Z 312.05,A -85,B 0,C 180,E1 -14359.753,E2 -14359.753} C_VEL
LIN {X 0,Y 340.698,Z 312.044,A -85,B 0,C 180,E1 -14362.32,E2 -14362.32} C_VEL
LIN {X 0,Y 340.017,Z 312.132,A -85,B 0,C 180,E1 -14363.306,E2 -14363.306} C_VEL
LIN {X 0,Y 337.178,Z 312.487,A -85,B 0,C 180,E1 -14364.911,E2 -14364.911} C_VEL
LIN {X 0,Y 334.775,Z 312.789,A -85,B 0,C 180,E1 -14366.211,E2 -14366.211} C_VEL
LIN {X 0,Y 333.731,Z 312.917,A -85,B 0,C 180,E1 -14367.216,E2 -14367.216} C_VEL
LIN {X 0,Y 333.639,Z 312.926,A -85,B 0,C 180,E1 -14367.557,E2 -14367.557} C_VEL
LIN {X 0,Y 333.714,Z 312.915,A -85,B 0,C 180,E1 -14371.028,E2 -14371.028} C_VEL
LIN {X 0,Y 333.738,Z 312.913,A -85,B 0,C 180,E1 -14373.754,E2 -14373.754} C_VEL
LIN {X 0,Y 333.659,Z 312.922,A -85,B 0,C 180,E1 -14377.72,E2 -14377.72} C_VEL
LIN {X 0,Y 333.744,Z 312.912,A -85,B 0,C 180,E1 -14381.587,E2 -14381.587} C_VEL
LIN {X 0,Y 333.812,Z 312.903,A -85,B 0,C 180,E1 -14385.577,E2 -14385.577} C_VEL
LIN {X 0,Y 333.822,Z 312.905,A -85,B 0,C 180,E1 -14389.078,E2 -14389.078} C_VEL
LIN {X 0,Y 333.999,Z 312.881,A -85,B 0,C 180,E1 -14392.747,E2 -14392.747} C_VEL
LIN {X 0,Y 333.806,Z 312.906,A -85,B 0,C 180,E1 -14395.169,E2 -14395.169} C_VEL
LIN {X 0,Y 334.106,Z 312.865,A -85,B 0,C 180,E1 -14397.589,E2 -14397.589} C_VEL
LIN {X 0,Y 334.23,Z 312.849,A -85,B 0,C 180,E1 -14400,E2 -14400} C_VEL
LIN {X 0,Y 334.097,Z 312.867,A -85,B 0,C 180,E1 -14402.411,E2 -14402.411} C_VEL
LIN {X 0,Y 334.001,Z 312.878,A -85,B 0,C 180,E1 -14406.039,E2 -14406.039} C_VEL
LIN {X 0,Y 333.824,Z 312.899,A -85,B 0,C 180,E1 -14409.696,E2 -14409.696} C_VEL
LIN {X 0,Y 333.801,Z 312.903,A -85,B 0,C 180,E1 -14413.391,E2 -14413.391} C_VEL
LIN {X 0,Y 333.723,Z 312.913,A -85,B 0,C 180,E1 -14417.148,E2 -14417.148} C_VEL
LIN {X 0,Y 333.689,Z 312.917,A -85,B 0,C 180,E1 -14419.693,E2 -14419.693} C_VEL
LIN {X 0,Y 333.671,Z 312.919,A -85,B 0,C 180,E1 -14423.59,E2 -14423.59} C_VEL
LIN {X 0,Y 333.679,Z 312.923,A -85,B 0,C 180,E1 -14426.251,E2 -14426.251} C_VEL
LIN {X 0,Y 333.663,Z 312.924,A -85,B 0,C 180,E1 -14430.366,E2 -14430.366} C_VEL
LIN {X 0,Y 333.642,Z 312.922,A -85,B 0,C 180,E1 -14433.208,E2 -14433.208} C_VEL
LIN {X 0,Y 333.668,Z 312.919,A -85,B 0,C 180,E1 -14436.832,E2 -14436.832} C_VEL
LIN {X 0,Y 333.649,Z 312.926,A -85,B 0,C 180,E1 -14440.767,E2 -14440.767} C_VEL
LIN {X 0,Y 333.648,Z 312.969,A -85,B 0,C 180,E1 -14444.163,E2 -14444.163} C_VEL
LIN {X 0,Y 334.807,Z 319.01,A -85,B 0,C 180,E1 -14447.8,E2 -14447.8} C_VEL
LIN {X 0,Y 335.839,Z 324.828,A -85,B 0,C 180,E1 -14451.112,E2 -14451.112} C_VEL
LIN {X 0,Y 336.301,Z 329.13,A -85,B 0,C 180,E1 -14453.445,E2 -14453.445} C_VEL
LIN {X 0,Y 335.653,Z 334.727,A -85,B 0,C 180,E1 -14456.299,E2 -14456.299} C_VEL
LIN {X 0,Y 334.565,Z 343.04,A -85,B 0,C 180,E1 -14460.419,E2 -14460.419} C_VEL
LIN {X 0,Y 333.784,Z 349.958,A -85,B 0,C 180,E1 -14463.758,E2 -14463.758} C_VEL
LIN {X 0,Y 333.059,Z 358.182,A -85,B 0,C 180,E1 -14467.677,E2 -14467.677} C_VEL
LIN {X 0,Y 332.894,Z 361.091,A -85,B 0,C 180,E1 -14469.048,E2 -14469.048} C_VEL
LIN {X 0,Y 335.016,Z 376.484,A -85,B 0,C 180,E1 -14469.815,E2 -14469.815} C_VEL
LIN {X 0,Y 336.4,Z 389.492,A -85,B 0,C 180,E1 -14470.692,E2 -14470.692} C_VEL
LIN {X 0,Y 337.271,Z 400.598,A -85,B 0,C 180,E1 -14471.638,E2 -14471.638} C_VEL
LIN {X 0,Y 337.282,Z 406.932,A -85,B 0,C 180,E1 -14472.257,E2 -14472.257} C_VEL
LIN {X 0,Y 336.046,Z 417.439,A -85,B 0,C 180,E1 -14473.444,E2 -14473.444} C_VEL
LIN {X 0,Y 334.964,Z 427.332,A -85,B 0,C 180,E1 -14474.828,E2 -14474.828} C_VEL
LIN {X 0,Y 334.117,Z 435.999,A -85,B 0,C 180,E1 -14476.312,E2 -14476.312} C_VEL
LIN {X 0,Y 333.391,Z 443.332,A -85,B 0,C 180,E1 -14477.83,E2 -14477.83} C_VEL
LIN {X 0,Y 332.739,Z 450.544,A -85,B 0,C 180,E1 -14479.657,E2 -14479.657} C_VEL
LIN {X 0,Y 332.398,Z 456.286,A -85,B 0,C 180,E1 -14481.489,E2 -14481.489} C_VEL
LIN {X 0,Y 332.245,Z 460.908,A -85,B 0,C 180,E1 -14483.38,E2 -14483.38} C_VEL
LIN {X 0,Y 332.239,Z 464.162,A -85,B 0,C 180,E1 -14485.146,E2 -14485.146} C_VEL
LIN {X 0,Y 332.199,Z 465.812,A -85,B 0,C 180,E1 -14486.361,E2 -14486.361} C_VEL
LIN {X 0,Y 332.377,Z 467.06,A -85,B 0,C 180,E1 -14487.576,E2 -14487.576} C_VEL
LIN {X 0,Y 332.401,Z 467.878,A -85,B 0,C 180,E1 -14488.789,E2 -14488.789} C_VEL
LIN {X 0,Y 332.409,Z 468.238,A -85,B 0,C 180,E1 -14490,E2 -14490} C_VEL
LIN {X 0,Y 332.381,Z 468.185,A -85,B 0,C 180,E1 -14491.212,E2 -14491.212} C_VEL
LIN {X 0,Y 332.315,Z 467.728,A -85,B 0,C 180,E1 -14492.424,E2 -14492.424} C_VEL
LIN {X 0,Y 332.167,Z 466.861,A -85,B 0,C 180,E1 -14493.639,E2 -14493.639} C_VEL
LIN {X 0,Y 332.104,Z 464.018,A -85,B 0,C 180,E1 -14495.945,E2 -14495.945} C_VEL
LIN {X 0,Y 332.265,Z 460.388,A -85,B 0,C 180,E1 -14497.903,E2 -14497.903} C_VEL
LIN {X 0,Y 332.588,Z 455.889,A -85,B 0,C 180,E1 -14499.733,E2 -14499.733} C_VEL
LIN {X 0,Y 333.298,Z 449.17,A -85,B 0,C 180,E1 -14501.864,E2 -14501.864} C_VEL
LIN {X 0,Y 334.35,Z 441.917,A -85,B 0,C 180,E1 -14503.679,E2 -14503.679} C_VEL
LIN {X 0,Y 335.587,Z 432.571,A -85,B 0,C 180,E1 -14505.559,E2 -14505.559} C_VEL
LIN {X 0,Y 336.99,Z 422.888,A -85,B 0,C 180,E1 -14507.133,E2 -14507.133} C_VEL
LIN {X 0,Y 338.751,Z 411.482,A -85,B 0,C 180,E1 -14508.602,E2 -14508.602} C_VEL
LIN {X 0,Y 339.318,Z 403.409,A -85,B 0,C 180,E1 -14509.498,E2 -14509.498} C_VEL
LIN {X 0,Y 339.017,Z 390.702,A -85,B 0,C 180,E1 -14510.723,E2 -14510.723} C_VEL
LIN {X 0,Y 337.634,Z 378.058,A -85,B 0,C 180,E1 -14511.771,E2 -14511.771} C_VEL
LIN {X 0,Y 335.22,Z 365.592,A -85,B 0,C 180,E1 -14512.66,E2 -14512.66} C_VEL
LIN {X 0,Y 333.295,Z 357.236,A -85,B 0,C 180,E1 -14513.196,E2 -14513.196} C_VEL
LIN {X 0,Y 334.156,Z 348.298,A -85,B 0,C 180,E1 -14517.562,E2 -14517.562} C_VEL
LIN {X 0,Y 335.169,Z 340.409,A -85,B 0,C 180,E1 -14521.616,E2 -14521.616} C_VEL
LIN {X 0,Y 336.02,Z 335.279,A -85,B 0,C 180,E1 -14524.383,E2 -14524.383} C_VEL
LIN {X 0,Y 336.651,Z 331.501,A -85,B 0,C 180,E1 -14526.511,E2 -14526.511} C_VEL
LIN {X 0,Y 336.551,Z 328.89,A -85,B 0,C 180,E1 -14528.089,E2 -14528.089} C_VEL
LIN {X 0,Y 335.825,Z 324.355,A -85,B 0,C 180,E1 -14531.115,E2 -14531.115} C_VEL
LIN {X 0,Y 334.97,Z 319.844,A -85,B 0,C 180,E1 -14534.491,E2 -14534.491} C_VEL
LIN {X 0,Y 334.237,Z 315.987,A -85,B 0,C 180,E1 -14537.711,E2 -14537.711} C_VEL
LIN {X 0,Y 333.65,Z 312.931,A -85,B 0,C 180,E1 -14540.808,E2 -14540.808} C_VEL
LIN {X 0,Y 333.68,Z 312.921,A -85,B 0,C 180,E1 -14543.861,E2 -14543.861} C_VEL
LIN {X 0,Y 333.649,Z 312.926,A -85,B 0,C 180,E1 -14547.412,E2 -14547.412} C_VEL
LIN {X 0,Y 333.715,Z 312.917,A -85,B 0,C 180,E1 -14551.028,E2 -14551.028} C_VEL
LIN {X 0,Y 333.74,Z 312.914,A -85,B 0,C 180,E1 -14553.754,E2 -14553.754} C_VEL
LIN {X 0,Y 333.723,Z 312.913,A -85,B 0,C 180,E1 -14557.914,E2 -14557.914} C_VEL
LIN {X 0,Y 333.799,Z 312.906,A -85,B 0,C 180,E1 -14561.59,E2 -14561.59} C_VEL
LIN {X 0,Y 333.812,Z 312.906,A -85,B 0,C 180,E1 -14565.576,E2 -14565.576} C_VEL
LIN {X 0,Y 333.822,Z 312.901,A -85,B 0,C 180,E1 -14569.077,E2 -14569.077} C_VEL
LIN {X 0,Y 333.972,Z 312.885,A -85,B 0,C 180,E1 -14572.746,E2 -14572.746} C_VEL
LIN {X 0,Y 333.806,Z 312.904,A -85,B 0,C 180,E1 -14575.169,E2 -14575.169} C_VEL
LIN {X 0,Y 334.109,Z 312.867,A -85,B 0,C 180,E1 -14577.589,E2 -14577.589} C_VEL
LIN {X 0,Y 334.251,Z 312.852,A -85,B 0,C 180,E1 -14580,E2 -14580} C_VEL
LIN {X 0,Y 334.111,Z 312.868,A -85,B 0,C 180,E1 -14582.411,E2 -14582.411} C_VEL
LIN {X 0,Y 333.971,Z 312.884,A -85,B 0,C 180,E1 -14586.52,E2 -14586.52} C_VEL
LIN {X 0,Y 333.968,Z 312.887,A -85,B 0,C 180,E1 -14587.254,E2 -14587.254} C_VEL
LIN {X 0,Y 333.862,Z 315.284,A -85,B 0,C 180,E1 -14590.921,E2 -14590.921} C_VEL
LIN {X 0,Y 333.646,Z 318.154,A -85,B 0,C 180,E1 -14594.922,E2 -14594.922} C_VEL
LIN {X 0,Y 333.685,Z 318.478,A -85,B 0,C 180,E1 -14595.026,E2 -14595.026} C_VEL
LIN {X 0,Y 338.98,Z 332.422,A -85,B 0,C 180,E1 -14596.254,E2 -14596.254} C_VEL
LIN {X 0,Y 342.16,Z 343.357,A -85,B 0,C 180,E1 -14597.327,E2 -14597.327} C_VEL
LIN {X 0,Y 343.068,Z 347.24,A -85,B 0,C 180,E1 -14597.741,E2 -14597.741} C_VEL
LIN {X 0,Y 342.26,Z 356.605,A -85,B 0,C 180,E1 -14598.598,E2 -14598.598} C_VEL
LIN {X 0,Y 340.77,Z 368.24,A -85,B 0,C 180,E1 -14599.895,E2 -14599.895} C_VEL
LIN {X 0,Y 339.415,Z 378.097,A -85,B 0,C 180,E1 -14601.285,E2 -14601.285} C_VEL
LIN {X 0,Y 337.865,Z 387.709,A -85,B 0,C 180,E1 -14602.956,E2 -14602.956} C_VEL
LIN {X 0,Y 336.605,Z 395.632,A -85,B 0,C 180,E1 -14604.682,E2 -14604.682} C_VEL
LIN {X 0,Y 335.48,Z 402.095,A -85,B 0,C 180,E1 -14606.434,E2 -14606.434} C_VEL
LIN {X 0,Y 334.437,Z 407.936,A -85,B 0,C 180,E1 -14608.446,E2 -14608.446} C_VEL
LIN {X 0,Y 333.704,Z 412.162,A -85,B 0,C 180,E1 -14610.361,E2 -14610.361} C_VEL
LIN {X 0,Y 333.035,Z 415.44,A -85,B 0,C 180,E1 -14612.422,E2 -14612.422} C_VEL
LIN {X 0,Y 332.525,Z 417.66,A -85,B 0,C 180,E1 -14614.796,E2 -14614.796} C_VEL
LIN {X 0,Y 332.32,Z 418.324,A -85,B 0,C 180,E1 -14616.521,E2 -14616.521} C_VEL
LIN {X 0,Y 332.241,Z 418.076,A -85,B 0,C 180,E1 -14618.493,E2 -14618.493} C_VEL
LIN {X 0,Y 332.298,Z 416.819,A -85,B 0,C 180,E1 -14620.413,E2 -14620.413} C_VEL
LIN {X 0,Y 332.573,Z 414.195,A -85,B 0,C 180,E1 -14622.55,E2 -14622.55} C_VEL
LIN {X 0,Y 332.91,Z 411.345,A -85,B 0,C 180,E1 -14624.159,E2 -14624.159} C_VEL
LIN {X 0,Y 333.398,Z 406.435,A -85,B 0,C 180,E1 -14626.227,E2 -14626.227} C_VEL
LIN {X 0,Y 333.913,Z 401.139,A -85,B 0,C 180,E1 -14627.962,E2 -14627.962} C_VEL
LIN {X 0,Y 334.701,Z 394.29,A -85,B 0,C 180,E1 -14629.763,E2 -14629.763} C_VEL
LIN {X 0,Y 335.579,Z 386.364,A -85,B 0,C 180,E1 -14631.453,E2 -14631.453} C_VEL
LIN {X 0,Y 336.64,Z 376.674,A -85,B 0,C 180,E1 -14633.115,E2 -14633.115} C_VEL
LIN {X 0,Y 337.736,Z 366.357,A -85,B 0,C 180,E1 -14634.545,E2 -14634.545} C_VEL
LIN {X 0,Y 338.724,Z 354.693,A -85,B 0,C 180,E1 -14635.84,E2 -14635.84} C_VEL
LIN {X 0,Y 339.74,Z 343.034,A -85,B 0,C 180,E1 -14636.845,E2 -14636.845} C_VEL
LIN {X 0,Y 337.261,Z 331.418,A -85,B 0,C 180,E1 -14637.79,E2 -14637.79} C_VEL
LIN {X 0,Y 334.003,Z 318.669,A -85,B 0,C 180,E1 -14638.615,E2 -14638.615} C_VEL
LIN {X 0,Y 332.793,Z 314.122,A -85,B 0,C 180,E1 -14638.886,E2 -14638.886} C_VEL
LIN {X 0,Y 332.817,Z 313.077,A -85,B 0,C 180,E1 -14639.972,E2 -14639.972} C_VEL
LIN {X 0,Y 333.293,Z 312.968,A -85,B 0,C 180,E1 -14643.716,E2 -14643.716} C_VEL
LIN {X 0,Y 333.531,Z 312.936,A -85,B 0,C 180,E1 -14646.399,E2 -14646.399} C_VEL
LIN {X 0,Y 333.653,Z 312.925,A -85,B 0,C 180,E1 -14649.017,E2 -14649.017} C_VEL
LIN {X 0,Y 333.741,Z 312.912,A -85,B 0,C 180,E1 -14651.586,E2 -14651.586} C_VEL
LIN {X 0,Y 333.809,Z 312.903,A -85,B 0,C 180,E1 -14655.577,E2 -14655.577} C_VEL
LIN {X 0,Y 333.834,Z 312.903,A -85,B 0,C 180,E1 -14659.078,E2 -14659.078} C_VEL
LIN {X 0,Y 333.969,Z 312.886,A -85,B 0,C 180,E1 -14662.746,E2 -14662.746} C_VEL
LIN {X 0,Y 333.805,Z 312.905,A -85,B 0,C 180,E1 -14665.169,E2 -14665.169} C_VEL
LIN {X 0,Y 334.106,Z 312.865,A -85,B 0,C 180,E1 -14667.589,E2 -14667.589} C_VEL
LIN {X 0,Y 334.247,Z 312.847,A -85,B 0,C 180,E1 -14670,E2 -14670} C_VEL
LIN {X 0,Y 334.108,Z 312.867,A -85,B 0,C 180,E1 -14672.411,E2 -14672.411} C_VEL
LIN {X 0,Y 334,Z 312.879,A -85,B 0,C 180,E1 -14676.039,E2 -14676.039} C_VEL
LIN {X 0,Y 333.85,Z 312.897,A -85,B 0,C 180,E1 -14679.696,E2 -14679.696} C_VEL
LIN {X 0,Y 333.797,Z 312.903,A -85,B 0,C 180,E1 -14683.391,E2 -14683.391} C_VEL
LIN {X 0,Y 333.747,Z 312.91,A -85,B 0,C 180,E1 -14687.146,E2 -14687.146} C_VEL
LIN {X 0,Y 333.738,Z 312.911,A -85,B 0,C 180,E1 -14689.69,E2 -14689.69} C_VEL
LIN {X 0,Y 333.693,Z 312.921,A -85,B 0,C 180,E1 -14692.278,E2 -14692.278} C_VEL
LIN {X 0,Y 333.737,Z 312.916,A -85,B 0,C 180,E1 -14696.246,E2 -14696.246} C_VEL
LIN {X 0,Y 333.712,Z 312.914,A -85,B 0,C 180,E1 -14698.972,E2 -14698.972} C_VEL
LIN {X 0,Y 333.644,Z 312.923,A -85,B 0,C 180,E1 -14702.587,E2 -14702.587} C_VEL
LIN {X 0,Y 333.677,Z 312.922,A -85,B 0,C 180,E1 -14706.139,E2 -14706.139} C_VEL
LIN {X 0,Y 333.648,Z 312.922,A -85,B 0,C 180,E1 -14709.193,E2 -14709.193} C_VEL
LIN {X 0,Y 333.634,Z 312.924,A -85,B 0,C 180,E1 -14712.5,E2 -14712.5} C_VEL
LIN {X 0,Y 333.598,Z 312.932,A -85,B 0,C 180,E1 -14715.955,E2 -14715.955} C_VEL
LIN {X 0,Y 333.649,Z 312.923,A -85,B 0,C 180,E1 -14719.316,E2 -14719.316} C_VEL
LIN {X 0,Y 333.667,Z 312.921,A -85,B 0,C 180,E1 -14723.168,E2 -14723.168} C_VEL
LIN {X 0,Y 333.676,Z 312.921,A -85,B 0,C 180,E1 -14725.342,E2 -14725.342} C_VEL
LIN {X 0,Y 333.639,Z 312.926,A -85,B 0,C 180,E1 -14727.557,E2 -14727.557} C_VEL
LIN {X 0,Y 332.95,Z 313.009,A -85,B 0,C 180,E1 -14728.564,E2 -14728.564} C_VEL
LIN {X 0,Y 330.097,Z 313.364,A -85,B 0,C 180,E1 -14730.204,E2 -14730.204} C_VEL
LIN {X 0,Y 327.718,Z 313.665,A -85,B 0,C 180,E1 -14731.532,E2 -14731.532} C_VEL
LIN {X 0,Y 326.733,Z 313.783,A -85,B 0,C 180,E1 -14732.559,E2 -14732.559} C_VEL
LIN {X 0,Y 326.671,Z 313.792,A -85,B 0,C 180,E1 -14732.907,E2 -14732.907} C_VEL
LIN {X 0,Y 326.651,Z 313.794,A -85,B 0,C 180,E1 -14735.871,E2 -14735.871} C_VEL
LIN {X 0,Y 326.634,Z 313.796,A -85,B 0,C 180,E1 -14739.863,E2 -14739.863} C_VEL
LIN {X 0,Y 326.667,Z 313.791,A -85,B 0,C 180,E1 -14742.47,E2 -14742.47} C_VEL
LIN {X 0,Y 326.763,Z 313.779,A -85,B 0,C 180,E1 -14746.315,E2 -14746.315} C_VEL
LIN {X 0,Y 326.787,Z 313.776,A -85,B 0,C 180,E1 -14750.093,E2 -14750.093} C_VEL
LIN {X 0,Y 326.988,Z 313.751,A -85,B 0,C 180,E1 -14753.831,E2 -14753.831} C_VEL
LIN {X 0,Y 327.047,Z 313.745,A -85,B 0,C 180,E1 -14757.537,E2 -14757.537} C_VEL
LIN {X 0,Y 327.182,Z 313.727,A -85,B 0,C 180,E1 -14760,E2 -14760} C_VEL
LIN {X 0,Y 327.037,Z 313.747,A -85,B 0,C 180,E1 -14762.463,E2 -14762.463} C_VEL
LIN {X 0,Y 326.955,Z 313.756,A -85,B 0,C 180,E1 -14766.17,E2 -14766.17} C_VEL
LIN {X 0,Y 326.787,Z 313.776,A -85,B 0,C 180,E1 -14769.907,E2 -14769.907} C_VEL
LIN {X 0,Y 326.763,Z 313.779,A -85,B 0,C 180,E1 -14773.685,E2 -14773.685} C_VEL
LIN {X 0,Y 326.667,Z 313.791,A -85,B 0,C 180,E1 -14777.53,E2 -14777.53} C_VEL
LIN {X 0,Y 326.634,Z 313.798,A -85,B 0,C 180,E1 -14780.137,E2 -14780.137} C_VEL
LIN {X 0,Y 326.646,Z 313.797,A -85,B 0,C 180,E1 -14784.13,E2 -14784.13} C_VEL
LIN {X 0,Y 326.631,Z 313.801,A -85,B 0,C 180,E1 -14788.253,E2 -14788.253} C_VEL
LIN {X 0,Y 326.578,Z 313.802,A -85,B 0,C 180,E1 -14791.097,E2 -14791.097} C_VEL
LIN {X 0,Y 326.611,Z 313.802,A -85,B 0,C 180,E1 -14794.019,E2 -14794.019} C_VEL
LIN {X 0,Y 326.63,Z 313.796,A -85,B 0,C 180,E1 -14797.238,E2 -14797.238} C_VEL
LIN {X 0,Y 326.58,Z 313.805,A -85,B 0,C 180,E1 -14801.131,E2 -14801.131} C_VEL
LIN {X 0,Y 326.626,Z 313.997,A -85,B 0,C 180,E1 -14803.942,E2 -14803.942} C_VEL
LIN {X 0,Y 327.527,Z 318.682,A -85,B 0,C 180,E1 -14806.85,E2 -14806.85} C_VEL
LIN {X 0,Y 328.601,Z 324.648,A -85,B 0,C 180,E1 -14810.35,E2 -14810.35} C_VEL
LIN {X 0,Y 329.232,Z 328.898,A -85,B 0,C 180,E1 -14812.753,E2 -14812.753} C_VEL
LIN {X 0,Y 328.985,Z 332.713,A -85,B 0,C 180,E1 -14814.774,E2 -14814.774} C_VEL
LIN {X 0,Y 327.984,Z 339.652,A -85,B 0,C 180,E1 -14818.333,E2 -14818.333} C_VEL
LIN {X 0,Y 327.17,Z 346.549,A -85,B 0,C 180,E1 -14821.797,E2 -14821.797} C_VEL
LIN {X 0,Y 326.298,Z 354.762,A -85,B 0,C 180,E1 -14825.843,E2 -14825.843} C_VEL
LIN {X 0,Y 325.822,Z 360.67,A -85,B 0,C 180,E1 -14828.696,E2 -14828.696} C_VEL
LIN {X 0,Y 327.801,Z 374.781,A -85,B 0,C 180,E1 -14829.385,E2 -14829.385} C_VEL
LIN {X 0,Y 329.265,Z 387.631,A -85,B 0,C 180,E1 -14830.256,E2 -14830.256} C_VEL
LIN {X 0,Y 330.282,Z 400.687,A -85,B 0,C 180,E1 -14831.386,E2 -14831.386} C_VEL
LIN {X 0,Y 330.321,Z 407.005,A -85,B 0,C 180,E1 -14832.031,E2 -14832.031} C_VEL
LIN {X 0,Y 328.916,Z 418.567,A -85,B 0,C 180,E1 -14833.394,E2 -14833.394} C_VEL
LIN {X 0,Y 327.759,Z 428.627,A -85,B 0,C 180,E1 -14834.878,E2 -14834.878} C_VEL
LIN {X 0,Y 326.97,Z 436.618,A -85,B 0,C 180,E1 -14836.324,E2 -14836.324} C_VEL
LIN {X 0,Y 326.115,Z 445.005,A -85,B 0,C 180,E1 -14838.186,E2 -14838.186} C_VEL
LIN {X 0,Y 325.564,Z 451.764,A -85,B 0,C 180,E1 -14840.055,E2 -14840.055} C_VEL
LIN {X 0,Y 325.257,Z 457.146,A -85,B 0,C 180,E1 -14841.926,E2 -14841.926} C_VEL
LIN {X 0,Y 325.194,Z 461.321,A -85,B 0,C 180,E1 -14843.797,E2 -14843.797} C_VEL
LIN {X 0,Y 325.151,Z 463.496,A -85,B 0,C 180,E1 -14845.04,E2 -14845.04} C_VEL
LIN {X 0,Y 325.12,Z 465.171,A -85,B 0,C 180,E1 -14846.282,E2 -14846.282} C_VEL
LIN {X 0,Y 325.295,Z 466.441,A -85,B 0,C 180,E1 -14847.523,E2 -14847.523} C_VEL
LIN {X 0,Y 325.338,Z 467.285,A -85,B 0,C 180,E1 -14848.762,E2 -14848.762} C_VEL
LIN {X 0,Y 325.344,Z 467.684,A -85,B 0,C 180,E1 -14850,E2 -14850} C_VEL
LIN {X 0,Y 325.317,Z 467.651,A -85,B 0,C 180,E1 -14851.238,E2 -14851.238} C_VEL
LIN {X 0,Y 325.217,Z 467.208,A -85,B 0,C 180,E1 -14852.477,E2 -14852.477} C_VEL
LIN {X 0,Y 325.084,Z 466.364,A -85,B 0,C 180,E1 -14853.719,E2 -14853.719} C_VEL
LIN {X 0,Y 325.021,Z 463.821,A -85,B 0,C 180,E1 -14855.917,E2 -14855.917} C_VEL
LIN {X 0,Y 325.194,Z 459.992,A -85,B 0,C 180,E1 -14858.075,E2 -14858.075} C_VEL
LIN {X 0,Y 325.539,Z 455.556,A -85,B 0,C 180,E1 -14859.946,E2 -14859.946} C_VEL
LIN {X 0,Y 326.335,Z 448.906,A -85,B 0,C 180,E1 -14862.121,E2 -14862.121} C_VEL
LIN {X 0,Y 327.404,Z 441.741,A -85,B 0,C 180,E1 -14863.975,E2 -14863.975} C_VEL
LIN {X 0,Y 328.622,Z 433.166,A -85,B 0,C 180,E1 -14865.765,E2 -14865.765} C_VEL
LIN {X 0,Y 330.042,Z 423.868,A -85,B 0,C 180,E1 -14867.345,E2 -14867.345} C_VEL
LIN {X 0,Y 331.873,Z 412.96,A -85,B 0,C 180,E1 -14868.841,E2 -14868.841} C_VEL
LIN {X 0,Y 332.594,Z 405.083,A -85,B 0,C 180,E1 -14869.761,E2 -14869.761} C_VEL
LIN {X 0,Y 332.478,Z 393.966,A -85,B 0,C 180,E1 -14870.926,E2 -14870.926} C_VEL
LIN {X 0,Y 331.612,Z 383.27,A -85,B 0,C 180,E1 -14871.894,E2 -14871.894} C_VEL
LIN {X 0,Y 329.656,Z 370.975,A -85,B 0,C 180,E1 -14872.869,E2 -14872.869} C_VEL
LIN {X 0,Y 326.807,Z 359.129,A -85,B 0,C 180,E1 -14873.708,E2 -14873.708} C_VEL
LIN {X 0,Y 326.33,Z 356.623,A -85,B 0,C 180,E1 -14873.853,E2 -14873.853} C_VEL
LIN {X 0,Y 327.086,Z 349.341,A -85,B 0,C 180,E1 -14877.514,E2 -14877.514} C_VEL
LIN {X 0,Y 327.933,Z 342.715,A -85,B 0,C 180,E1 -14880.99,E2 -14880.99} C_VEL
LIN {X 0,Y 329.033,Z 336.376,A -85,B 0,C 180,E1 -14884.474,E2 -14884.474} C_VEL
LIN {X 0,Y 329.701,Z 332.617,A -85,B 0,C 180,E1 -14886.645,E2 -14886.645} C_VEL
LIN {X 0,Y 329.404,Z 328.976,A -85,B 0,C 180,E1 -14888.978,E2 -14888.978} C_VEL
LIN {X 0,Y 328.56,Z 324.177,A -85,B 0,C 180,E1 -14892.36,E2 -14892.36} C_VEL
LIN {X 0,Y 327.922,Z 320.788,A -85,B 0,C 180,E1 -14895.012,E2 -14895.012} C_VEL
LIN {X 0,Y 327.15,Z 316.6,A -85,B 0,C 180,E1 -14898.755,E2 -14898.755} C_VEL
LIN {X 0,Y 326.596,Z 313.805,A -85,B 0,C 180,E1 -14901.76,E2 -14901.76} C_VEL
LIN {X 0,Y 326.623,Z 313.799,A -85,B 0,C 180,E1 -14904.851,E2 -14904.851} C_VEL
LIN {X 0,Y 326.613,Z 313.802,A -85,B 0,C 180,E1 -14907.456,E2 -14907.456} C_VEL
LIN {X 0,Y 326.664,Z 313.796,A -85,B 0,C 180,E1 -14910.341,E2 -14910.341} C_VEL
LIN {X 0,Y 326.694,Z 313.792,A -85,B 0,C 180,E1 -14914.516,E2 -14914.516} C_VEL
LIN {X 0,Y 326.653,Z 313.797,A -85,B 0,C 180,E1 -14918.546,E2 -14918.546} C_VEL
LIN {X 0,Y 326.748,Z 313.786,A -85,B 0,C 180,E1 -14921.178,E2 -14921.178} C_VEL
LIN {X 0,Y 326.767,Z 313.784,A -85,B 0,C 180,E1 -14925.433,E2 -14925.433} C_VEL
LIN {X 0,Y 326.763,Z 313.78,A -85,B 0,C 180,E1 -14928.839,E2 -14928.839} C_VEL
LIN {X 0,Y 326.927,Z 313.763,A -85,B 0,C 180,E1 -14932.589,E2 -14932.589} C_VEL
LIN {X 0,Y 326.772,Z 313.78,A -85,B 0,C 180,E1 -14935.065,E2 -14935.065} C_VEL
LIN {X 0,Y 327.049,Z 313.746,A -85,B 0,C 180,E1 -14937.537,E2 -14937.537} C_VEL
LIN {X 0,Y 327.202,Z 313.73,A -85,B 0,C 180,E1 -14940,E2 -14940} C_VEL
LIN {X 0,Y 327.052,Z 313.747,A -85,B 0,C 180,E1 -14942.463,E2 -14942.463} C_VEL
LIN {X 0,Y 326.95,Z 313.892,A -85,B 0,C 180,E1 -14946.52,E2 -14946.52} C_VEL
LIN {X 0,Y 326.963,Z 315.017,A -85,B 0,C 180,E1 -14948.654,E2 -14948.654} C_VEL
LIN {X 0,Y 326.772,Z 317.544,A -85,B 0,C 180,E1 -14952.42,E2 -14952.42} C_VEL
LIN {X 0,Y 326.708,Z 318.884,A -85,B 0,C 180,E1 -14954.331,E2 -14954.331} C_VEL
LIN {X 0,Y 327.843,Z 322.005,A -85,B 0,C 180,E1 -14954.594,E2 -14954.594} C_VEL
LIN {X 0,Y 332.585,Z 334.299,A -85,B 0,C 180,E1 -14955.77,E2 -14955.77} C_VEL
LIN {X 0,Y 335.665,Z 345.1,A -85,B 0,C 180,E1 -14956.888,E2 -14956.888} C_VEL
LIN {X 0,Y 336.64,Z 349.407,A -85,B 0,C 180,E1 -14957.366,E2 -14957.366} C_VEL
LIN {X 0,Y 335.317,Z 361.366,A -85,B 0,C 180,E1 -14958.539,E2 -14958.539} C_VEL
LIN {X 0,Y 333.836,Z 371.983,A -85,B 0,C 180,E1 -14959.844,E2 -14959.844} C_VEL
LIN {X 0,Y 332.382,Z 381.467,A -85,B 0,C 180,E1 -14961.292,E2 -14961.292} C_VEL
LIN {X 0,Y 330.709,Z 390.988,A -85,B 0,C 180,E1 -14963.109,E2 -14963.109} C_VEL
LIN {X 0,Y 329.384,Z 398.591,A -85,B 0,C 180,E1 -14964.923,E2 -14964.923} C_VEL
LIN {X 0,Y 328.273,Z 404.624,A -85,B 0,C 180,E1 -14966.717,E2 -14966.717} C_VEL
LIN {X 0,Y 327.205,Z 410.342,A -85,B 0,C 180,E1 -14968.931,E2 -14968.931} C_VEL
LIN {X 0,Y 326.384,Z 414.467,A -85,B 0,C 180,E1 -14971.117,E2 -14971.117} C_VEL
LIN {X 0,Y 325.888,Z 416.621,A -85,B 0,C 180,E1 -14972.747,E2 -14972.747} C_VEL
LIN {X 0,Y 325.467,Z 418.345,A -85,B 0,C 180,E1 -14974.859,E2 -14974.859} C_VEL
LIN {X 0,Y 325.184,Z 418.915,A -85,B 0,C 180,E1 -14977.239,E2 -14977.239} C_VEL
LIN {X 0,Y 325.155,Z 418.397,A -85,B 0,C 180,E1 -14978.911,E2 -14978.911} C_VEL
LIN {X 0,Y 325.271,Z 416.886,A -85,B 0,C 180,E1 -14980.866,E2 -14980.866} C_VEL
LIN {X 0,Y 325.551,Z 414.409,A -85,B 0,C 180,E1 -14982.777,E2 -14982.777} C_VEL
LIN {X 0,Y 325.921,Z 410.997,A -85,B 0,C 180,E1 -14984.635,E2 -14984.635} C_VEL
LIN {X 0,Y 326.372,Z 406.637,A -85,B 0,C 180,E1 -14986.442,E2 -14986.442} C_VEL
LIN {X 0,Y 326.936,Z 401.265,A -85,B 0,C 180,E1 -14988.21,E2 -14988.21} C_VEL
LIN {X 0,Y 327.706,Z 394.709,A -85,B 0,C 180,E1 -14989.955,E2 -14989.955} C_VEL
LIN {X 0,Y 328.625,Z 386.811,A -85,B 0,C 180,E1 -14991.669,E2 -14991.669} C_VEL
LIN {X 0,Y 329.721,Z 377.147,A -85,B 0,C 180,E1 -14993.357,E2 -14993.357} C_VEL
LIN {X 0,Y 330.903,Z 366.229,A -85,B 0,C 180,E1 -14994.894,E2 -14994.894} C_VEL
LIN {X 0,Y 331.907,Z 354.567,A -85,B 0,C 180,E1 -14996.194,E2 -14996.194} C_VEL
LIN {X 0,Y 332.817,Z 344.786,A -85,B 0,C 180,E1 -14997.06,E2 -14997.06} C_VEL
LIN {X 0,Y 331.64,Z 338.031,A -85,B 0,C 180,E1 -14997.65,E2 -14997.65} C_VEL
LIN {X 0,Y 328.545,Z 325.166,A -85,B 0,C 180,E1 -14998.617,E2 -14998.617} C_VEL
LIN {X 0,Y 325.746,Z 314.6,A -85,B 0,C 180,E1 -14999.26,E2 -14999.26} C_VEL
LIN {X 0,Y 325.79,Z 313.903,A -85,B 0,C 180,E1 -15000.253,E2 -15000.253} C_VEL
LIN {X 0,Y 326.16,Z 313.858,A -85,B 0,C 180,E1 -15003.095,E2 -15003.095} C_VEL
LIN {X 0,Y 326.433,Z 313.821,A -85,B 0,C 180,E1 -15005.854,E2 -15005.854} C_VEL
LIN {X 0,Y 326.6,Z 313.8,A -85,B 0,C 180,E1 -15008.542,E2 -15008.542} C_VEL
LIN {X 0,Y 326.665,Z 313.792,A -85,B 0,C 180,E1 -15012.47,E2 -15012.47} C_VEL
LIN {X 0,Y 326.76,Z 313.78,A -85,B 0,C 180,E1 -15016.315,E2 -15016.315} C_VEL
LIN {X 0,Y 326.805,Z 313.774,A -85,B 0,C 180,E1 -15020.093,E2 -15020.093} C_VEL
LIN {X 0,Y 326.953,Z 313.755,A -85,B 0,C 180,E1 -15023.83,E2 -15023.83} C_VEL
LIN {X 0,Y 327.046,Z 313.744,A -85,B 0,C 180,E1 -15027.537,E2 -15027.537} C_VEL
LIN {X 0,Y 327.198,Z 313.725,A -85,B 0,C 180,E1 -15030,E2 -15030} C_VEL
LIN {X 0,Y 327.048,Z 313.747,A -85,B 0,C 180,E1 -15032.463,E2 -15032.463} C_VEL
LIN {X 0,Y 326.953,Z 313.757,A -85,B 0,C 180,E1 -15036.17,E2 -15036.17} C_VEL
LIN {X 0,Y 326.805,Z 313.774,A -85,B 0,C 180,E1 -15039.907,E2 -15039.907} C_VEL
LIN {X 0,Y 326.76,Z 313.78,A -85,B 0,C 180,E1 -15043.685,E2 -15043.685} C_VEL
LIN {X 0,Y 326.7,Z 313.787,A -85,B 0,C 180,E1 -15047.528,E2 -15047.528} C_VEL
LIN {X 0,Y 326.664,Z 313.795,A -85,B 0,C 180,E1 -15050.135,E2 -15050.135} C_VEL
LIN {X 0,Y 326.653,Z 313.797,A -85,B 0,C 180,E1 -15054.129,E2 -15054.129} C_VEL
LIN {X 0,Y 326.686,Z 313.789,A -85,B 0,C 180,E1 -15056.858,E2 -15056.858} C_VEL
LIN {X 0,Y 326.64,Z 313.796,A -85,B 0,C 180,E1 -15060.611,E2 -15060.611} C_VEL
LIN {X 0,Y 326.608,Z 313.804,A -85,B 0,C 180,E1 -15064.02,E2 -15064.02} C_VEL
LIN {X 0,Y 326.629,Z 313.796,A -85,B 0,C 180,E1 -15067.239,E2 -15067.239} C_VEL
LIN {X 0,Y 326.579,Z 313.802,A -85,B 0,C 180,E1 -15071.132,E2 -15071.132} C_VEL
LIN {X 0,Y 326.529,Z 313.808,A -85,B 0,C 180,E1 -15074.743,E2 -15074.743} C_VEL
LIN {X 0,Y 326.578,Z 313.804,A -85,B 0,C 180,E1 -15078.155,E2 -15078.155} C_VEL
LIN {X 0,Y 326.626,Z 313.799,A -85,B 0,C 180,E1 -15081.392,E2 -15081.392} C_VEL
LIN {X 0,Y 326.621,Z 313.797,A -85,B 0,C 180,E1 -15084.852,E2 -15084.852} C_VEL
LIN {X 0,Y 326.603,Z 313.803,A -85,B 0,C 180,E1 -15087.542,E2 -15087.542} C_VEL
LIN {X 0,Y 326.663,Z 313.792,A -85,B 0,C 180,E1 -15090.341,E2 -15090.341} C_VEL
LIN {X 0,Y 326.671,Z 313.792,A -85,B 0,C 180,E1 -15092.907,E2 -15092.907} C_VEL
LIN {X 0,Y 326.045,Z 313.874,A -85,B 0,C 180,E1 -15093.936,E2 -15093.936} C_VEL
LIN {X 0,Y 323.179,Z 314.232,A -85,B 0,C 180,E1 -15095.608,E2 -15095.608} C_VEL
LIN {X 0,Y 320.715,Z 314.535,A -85,B 0,C 180,E1 -15096.963,E2 -15096.963} C_VEL
LIN {X 0,Y 319.648,Z 314.666,A -85,B 0,C 180,E1 -15098.013,E2 -15098.013} C_VEL
LIN {X 0,Y 319.559,Z 314.676,A -85,B 0,C 180,E1 -15098.369,E2 -15098.369} C_VEL
LIN {X 0,Y 319.627,Z 314.668,A -85,B 0,C 180,E1 -15102.071,E2 -15102.071} C_VEL
LIN {X 0,Y 319.735,Z 314.654,A -85,B 0,C 180,E1 -15106.008,E2 -15106.008} C_VEL
LIN {X 0,Y 319.739,Z 314.654,A -85,B 0,C 180,E1 -15109.872,E2 -15109.872} C_VEL
LIN {X 0,Y 319.942,Z 314.629,A -85,B 0,C 180,E1 -15113.694,E2 -15113.694} C_VEL
LIN {X 0,Y 319.99,Z 314.624,A -85,B 0,C 180,E1 -15117.483,E2 -15117.483} C_VEL
LIN {X 0,Y 320.134,Z 314.605,A -85,B 0,C 180,E1 -15120,E2 -15120} C_VEL
LIN {X 0,Y 319.981,Z 314.626,A -85,B 0,C 180,E1 -15122.518,E2 -15122.518} C_VEL
LIN {X 0,Y 319.912,Z 314.634,A -85,B 0,C 180,E1 -15126.306,E2 -15126.306} C_VEL
LIN {X 0,Y 319.739,Z 314.655,A -85,B 0,C 180,E1 -15130.128,E2 -15130.128} C_VEL
LIN {X 0,Y 319.736,Z 314.655,A -85,B 0,C 180,E1 -15133.992,E2 -15133.992} C_VEL
LIN {X 0,Y 319.628,Z 314.669,A -85,B 0,C 180,E1 -15137.929,E2 -15137.929} C_VEL
LIN {X 0,Y 319.571,Z 314.676,A -85,B 0,C 180,E1 -15141.954,E2 -15141.954} C_VEL
LIN {X 0,Y 319.582,Z 314.676,A -85,B 0,C 180,E1 -15146.093,E2 -15146.093} C_VEL
LIN {X 0,Y 319.561,Z 314.677,A -85,B 0,C 180,E1 -15148.937,E2 -15148.937} C_VEL
LIN {X 0,Y 319.529,Z 314.682,A -85,B 0,C 180,E1 -15151.862,E2 -15151.862} C_VEL
LIN {X 0,Y 319.583,Z 314.674,A -85,B 0,C 180,E1 -15155.543,E2 -15155.543} C_VEL
LIN {X 0,Y 319.575,Z 314.679,A -85,B 0,C 180,E1 -15158.008,E2 -15158.008} C_VEL
LIN {X 0,Y 319.528,Z 314.684,A -85,B 0,C 180,E1 -15161.597,E2 -15161.597} C_VEL
LIN {X 0,Y 319.557,Z 314.773,A -85,B 0,C 180,E1 -15163.571,E2 -15163.571} C_VEL
LIN {X 0,Y 320.655,Z 320.52,A -85,B 0,C 180,E1 -15167.199,E2 -15167.199} C_VEL
LIN {X 0,Y 321.687,Z 326.34,A -85,B 0,C 180,E1 -15170.685,E2 -15170.685} C_VEL
LIN {X 0,Y 322.237,Z 330.644,A -85,B 0,C 180,E1 -15173.147,E2 -15173.147} C_VEL
LIN {X 0,Y 321.559,Z 336.271,A -85,B 0,C 180,E1 -15176.154,E2 -15176.154} C_VEL
LIN {X 0,Y 320.428,Z 344.513,A -85,B 0,C 180,E1 -15180.429,E2 -15180.429} C_VEL
LIN {X 0,Y 319.498,Z 352.353,A -85,B 0,C 180,E1 -15184.407,E2 -15184.407} C_VEL
LIN {X 0,Y 318.808,Z 360.129,A -85,B 0,C 180,E1 -15188.288,E2 -15188.288} C_VEL
LIN {X 0,Y 320.934,Z 375.519,A -85,B 0,C 180,E1 -15189.091,E2 -15189.091} C_VEL
LIN {X 0,Y 322.417,Z 389.16,A -85,B 0,C 180,E1 -15190.069,E2 -15190.069} C_VEL
LIN {X 0,Y 323.297,Z 400.862,A -85,B 0,C 180,E1 -15191.134,E2 -15191.134} C_VEL
LIN {X 0,Y 323.366,Z 407.074,A -85,B 0,C 180,E1 -15191.794,E2 -15191.794} C_VEL
LIN {X 0,Y 321.933,Z 418.529,A -85,B 0,C 180,E1 -15193.186,E2 -15193.186} C_VEL
LIN {X 0,Y 320.699,Z 428.78,A -85,B 0,C 180,E1 -15194.753,E2 -15194.753} C_VEL
LIN {X 0,Y 319.827,Z 437.156,A -85,B 0,C 180,E1 -15196.336,E2 -15196.336} C_VEL
LIN {X 0,Y 318.98,Z 445.355,A -85,B 0,C 180,E1 -15198.241,E2 -15198.241} C_VEL
LIN {X 0,Y 318.518,Z 450.937,A -85,B 0,C 180,E1 -15199.833,E2 -15199.833} C_VEL
LIN {X 0,Y 318.194,Z 456.379,A -85,B 0,C 180,E1 -15201.746,E2 -15201.746} C_VEL
LIN {X 0,Y 318.104,Z 460.942,A -85,B 0,C 180,E1 -15203.83,E2 -15203.83} C_VEL
LIN {X 0,Y 318.069,Z 462.821,A -85,B 0,C 180,E1 -15204.929,E2 -15204.929} C_VEL
LIN {X 0,Y 318.044,Z 464.531,A -85,B 0,C 180,E1 -15206.199,E2 -15206.199} C_VEL
LIN {X 0,Y 318.199,Z 465.82,A -85,B 0,C 180,E1 -15207.468,E2 -15207.468} C_VEL
LIN {X 0,Y 318.276,Z 466.688,A -85,B 0,C 180,E1 -15208.735,E2 -15208.735} C_VEL
LIN {X 0,Y 318.28,Z 467.129,A -85,B 0,C 180,E1 -15210,E2 -15210} C_VEL
LIN {X 0,Y 318.253,Z 467.115,A -85,B 0,C 180,E1 -15211.265,E2 -15211.265} C_VEL
LIN {X 0,Y 318.12,Z 466.69,A -85,B 0,C 180,E1 -15212.532,E2 -15212.532} C_VEL
LIN {X 0,Y 318.005,Z 465.869,A -85,B 0,C 180,E1 -15213.802,E2 -15213.802} C_VEL
LIN {X 0,Y 317.927,Z 463.633,A -85,B 0,C 180,E1 -15215.868,E2 -15215.868} C_VEL
LIN {X 0,Y 318.05,Z 460.839,A -85,B 0,C 180,E1 -15217.619,E2 -15217.619} C_VEL
LIN {X 0,Y 318.343,Z 456.813,A -85,B 0,C 180,E1 -15219.531,E2 -15219.531} C_VEL
LIN {X 0,Y 318.892,Z 451.669,A -85,B 0,C 180,E1 -15221.441,E2 -15221.441} C_VEL
LIN {X 0,Y 319.911,Z 445.275,A -85,B 0,C 180,E1 -15223.337,E2 -15223.337} C_VEL
LIN {X 0,Y 321.171,Z 437.416,A -85,B 0,C 180,E1 -15225.224,E2 -15225.224} C_VEL
LIN {X 0,Y 322.602,Z 427.695,A -85,B 0,C 180,E1 -15227.104,E2 -15227.104} C_VEL
LIN {X 0,Y 324.371,Z 417.795,A -85,B 0,C 180,E1 -15228.638,E2 -15228.638} C_VEL
LIN {X 0,Y 325.771,Z 408.216,A -85,B 0,C 180,E1 -15229.864,E2 -15229.864} C_VEL
LIN {X 0,Y 325.934,Z 397.598,A -85,B 0,C 180,E1 -15231.069,E2 -15231.069} C_VEL
LIN {X 0,Y 325.208,Z 385.858,A -85,B 0,C 180,E1 -15232.217,E2 -15232.217} C_VEL
LIN {X 0,Y 323.725,Z 374.845,A -85,B 0,C 180,E1 -15233.172,E2 -15233.172} C_VEL
LIN {X 0,Y 320.969,Z 362.305,A -85,B 0,C 180,E1 -15234.143,E2 -15234.143} C_VEL
LIN {X 0,Y 319.391,Z 355.921,A -85,B 0,C 180,E1 -15234.597,E2 -15234.597} C_VEL
LIN {X 0,Y 320.322,Z 348.158,A -85,B 0,C 180,E1 -15238.643,E2 -15238.643} C_VEL
LIN {X 0,Y 321.557,Z 339.997,A -85,B 0,C 180,E1 -15243.121,E2 -15243.121} C_VEL
LIN {X 0,Y 322.641,Z 334.543,A -85,B 0,C 180,E1 -15246.297,E2 -15246.297} C_VEL
LIN {X 0,Y 322.596,Z 331.34,A -85,B 0,C 180,E1 -15248.345,E2 -15248.345} C_VEL
LIN {X 0,Y 321.717,Z 326.149,A -85,B 0,C 180,E1 -15252.034,E2 -15252.034} C_VEL
LIN {X 0,Y 320.897,Z 321.851,A -85,B 0,C 180,E1 -15255.506,E2 -15255.506} C_VEL
LIN {X 0,Y 320.27,Z 318.25,A -85,B 0,C 180,E1 -15258.828,E2 -15258.828} C_VEL
LIN {X 0,Y 319.597,Z 314.677,A -85,B 0,C 180,E1 -15262.797,E2 -15262.797} C_VEL
LIN {X 0,Y 319.581,Z 314.678,A -85,B 0,C 180,E1 -15266.686,E2 -15266.686} C_VEL
LIN {X 0,Y 319.595,Z 314.676,A -85,B 0,C 180,E1 -15269.617,E2 -15269.617} C_VEL
LIN {X 0,Y 319.613,Z 314.674,A -85,B 0,C 180,E1 -15272.498,E2 -15272.498} C_VEL
LIN {X 0,Y 319.609,Z 314.67,A -85,B 0,C 180,E1 -15275.304,E2 -15275.304} C_VEL
LIN {X 0,Y 319.602,Z 314.672,A -85,B 0,C 180,E1 -15278.048,E2 -15278.048} C_VEL
LIN {X 0,Y 319.694,Z 314.664,A -85,B 0,C 180,E1 -15280.962,E2 -15280.962} C_VEL
LIN {X 0,Y 319.735,Z 314.658,A -85,B 0,C 180,E1 -15285.276,E2 -15285.276} C_VEL
LIN {X 0,Y 319.72,Z 314.658,A -85,B 0,C 180,E1 -15288.589,E2 -15288.589} C_VEL
LIN {X 0,Y 319.882,Z 314.641,A -85,B 0,C 180,E1 -15292.425,E2 -15292.425} C_VEL
LIN {X 0,Y 319.74,Z 314.656,A -85,B 0,C 180,E1 -15294.956,E2 -15294.956} C_VEL
LIN {X 0,Y 319.993,Z 314.625,A -85,B 0,C 180,E1 -15297.482,E2 -15297.482} C_VEL
LIN {X 0,Y 320.154,Z 314.608,A -85,B 0,C 180,E1 -15300,E2 -15300} C_VEL
LIN {X 0,Y 319.995,Z 314.626,A -85,B 0,C 180,E1 -15302.517,E2 -15302.517} C_VEL
LIN {X 0,Y 319.939,Z 314.872,A -85,B 0,C 180,E1 -15306.306,E2 -15306.306} C_VEL
LIN {X 0,Y 319.954,Z 316.407,A -85,B 0,C 180,E1 -15308.845,E2 -15308.845} C_VEL
LIN {X 0,Y 319.761,Z 318.947,A -85,B 0,C 180,E1 -15312.697,E2 -15312.697} C_VEL
LIN {X 0,Y 319.747,Z 319.557,A -85,B 0,C 180,E1 -15313.586,E2 -15313.586} C_VEL
LIN {X 0,Y 321.027,Z 322.875,A -85,B 0,C 180,E1 -15313.914,E2 -15313.914} C_VEL
LIN {X 0,Y 325.796,Z 335.085,A -85,B 0,C 180,E1 -15315.137,E2 -15315.137} C_VEL
LIN {X 0,Y 328.937,Z 345.55,A -85,B 0,C 180,E1 -15316.285,E2 -15316.285} C_VEL
LIN {X 0,Y 330.15,Z 351.942,A -85,B 0,C 180,E1 -15317.02,E2 -15317.02} C_VEL
LIN {X 0,Y 328.649,Z 363.698,A -85,B 0,C 180,E1 -15318.225,E2 -15318.225} C_VEL
LIN {X 0,Y 327.088,Z 374.216,A -85,B 0,C 180,E1 -15319.591,E2 -15319.591} C_VEL
LIN {X 0,Y 325.392,Z 384.174,A -85,B 0,C 180,E1 -15321.209,E2 -15321.209} C_VEL
LIN {X 0,Y 323.791,Z 393.012,A -85,B 0,C 180,E1 -15322.998,E2 -15322.998} C_VEL
LIN {X 0,Y 322.434,Z 400.153,A -85,B 0,C 180,E1 -15324.808,E2 -15324.808} C_VEL
LIN {X 0,Y 321.195,Z 406.351,A -85,B 0,C 180,E1 -15326.785,E2 -15326.785} C_VEL
LIN {X 0,Y 320.188,Z 411.424,A -85,B 0,C 180,E1 -15328.874,E2 -15328.874} C_VEL
LIN {X 0,Y 319.41,Z 415.072,A -85,B 0,C 180,E1 -15330.893,E2 -15330.893} C_VEL
LIN {X 0,Y 318.741,Z 417.763,A -85,B 0,C 180,E1 -15333.083,E2 -15333.083} C_VEL
LIN {X 0,Y 318.331,Z 419.167,A -85,B 0,C 180,E1 -15335.226,E2 -15335.226} C_VEL
LIN {X 0,Y 318.122,Z 419.437,A -85,B 0,C 180,E1 -15337.314,E2 -15337.314} C_VEL
LIN {X 0,Y 318.105,Z 418.308,A -85,B 0,C 180,E1 -15339.844,E2 -15339.844} C_VEL
LIN {X 0,Y 318.396,Z 415.645,A -85,B 0,C 180,E1 -15342.317,E2 -15342.317} C_VEL
LIN {X 0,Y 318.713,Z 412.88,A -85,B 0,C 180,E1 -15344.013,E2 -15344.013} C_VEL
LIN {X 0,Y 319.136,Z 408.997,A -85,B 0,C 180,E1 -15345.819,E2 -15345.819} C_VEL
LIN {X 0,Y 319.687,Z 404.121,A -85,B 0,C 180,E1 -15347.608,E2 -15347.608} C_VEL
LIN {X 0,Y 320.349,Z 398.099,A -85,B 0,C 180,E1 -15349.394,E2 -15349.394} C_VEL
LIN {X 0,Y 321.291,Z 390.225,A -85,B 0,C 180,E1 -15351.273,E2 -15351.273} C_VEL
LIN {X 0,Y 322.392,Z 381.055,A -85,B 0,C 180,E1 -15353.035,E2 -15353.035} C_VEL
LIN {X 0,Y 323.533,Z 371.043,A -85,B 0,C 180,E1 -15354.596,E2 -15354.596} C_VEL
LIN {X 0,Y 324.654,Z 360.323,A -85,B 0,C 180,E1 -15355.935,E2 -15355.935} C_VEL
LIN {X 0,Y 325.647,Z 348.67,A -85,B 0,C 180,E1 -15357.099,E2 -15357.099} C_VEL
LIN {X 0,Y 325.938,Z 345.35,A -85,B 0,C 180,E1 -15357.38,E2 -15357.38} C_VEL
LIN {X 0,Y 323.51,Z 333.665,A -85,B 0,C 180,E1 -15358.392,E2 -15358.392} C_VEL
LIN {X 0,Y 320.19,Z 320.745,A -85,B 0,C 180,E1 -15359.297,E2 -15359.297} C_VEL
LIN {X 0,Y 318.732,Z 315.116,A -85,B 0,C 180,E1 -15359.617,E2 -15359.617} C_VEL
LIN {X 0,Y 318.819,Z 314.772,A -85,B 0,C 180,E1 -15360.99,E2 -15360.99} C_VEL
LIN {X 0,Y 319.302,Z 314.709,A -85,B 0,C 180,E1 -15364.479,E2 -15364.479} C_VEL
LIN {X 0,Y 319.532,Z 314.68,A -85,B 0,C 180,E1 -15368.043,E2 -15368.043} C_VEL
LIN {X 0,Y 319.615,Z 314.669,A -85,B 0,C 180,E1 -15372.07,E2 -15372.07} C_VEL
LIN {X 0,Y 319.733,Z 314.655,A -85,B 0,C 180,E1 -15376.008,E2 -15376.008} C_VEL
LIN {X 0,Y 319.752,Z 314.652,A -85,B 0,C 180,E1 -15379.873,E2 -15379.873} C_VEL
LIN {X 0,Y 319.91,Z 314.633,A -85,B 0,C 180,E1 -15383.694,E2 -15383.694} C_VEL
LIN {X 0,Y 319.99,Z 314.623,A -85,B 0,C 180,E1 -15387.482,E2 -15387.482} C_VEL
LIN {X 0,Y 320.15,Z 314.603,A -85,B 0,C 180,E1 -15390,E2 -15390} C_VEL
LIN {X 0,Y 319.992,Z 314.626,A -85,B 0,C 180,E1 -15392.518,E2 -15392.518} C_VEL
LIN {X 0,Y 319.91,Z 314.635,A -85,B 0,C 180,E1 -15396.306,E2 -15396.306} C_VEL
LIN {X 0,Y 319.752,Z 314.654,A -85,B 0,C 180,E1 -15400.127,E2 -15400.127} C_VEL
LIN {X 0,Y 319.732,Z 314.658,A -85,B 0,C 180,E1 -15404.724,E2 -15404.724} C_VEL
LIN {X 0,Y 319.69,Z 314.661,A -85,B 0,C 180,E1 -15409.038,E2 -15409.038} C_VEL
LIN {X 0,Y 319.571,Z 314.675,A -85,B 0,C 180,E1 -15413.32,E2 -15413.32} C_VEL
LIN {X 0,Y 319.636,Z 314.671,A -85,B 0,C 180,E1 -15416.088,E2 -15416.088} C_VEL
LIN {X 0,Y 319.59,Z 314.673,A -85,B 0,C 180,E1 -15418.934,E2 -15418.934} C_VEL
LIN {X 0,Y 319.533,Z 314.683,A -85,B 0,C 180,E1 -15421.862,E2 -15421.862} C_VEL
LIN {X 0,Y 319.581,Z 314.675,A -85,B 0,C 180,E1 -15425.543,E2 -15425.543} C_VEL
LIN {X 0,Y 319.574,Z 314.68,A -85,B 0,C 180,E1 -15428.008,E2 -15428.008} C_VEL
LIN {X 0,Y 319.527,Z 314.683,A -85,B 0,C 180,E1 -15431.597,E2 -15431.597} C_VEL
LIN {X 0,Y 319.49,Z 314.686,A -85,B 0,C 180,E1 -15435.258,E2 -15435.258} C_VEL
LIN {X 0,Y 319.53,Z 314.68,A -85,B 0,C 180,E1 -15438.712,E2 -15438.712} C_VEL
LIN {X 0,Y 319.563,Z 314.676,A -85,B 0,C 180,E1 -15442.348,E2 -15442.348} C_VEL
LIN {X 0,Y 319.562,Z 314.677,A -85,B 0,C 180,E1 -15445.124,E2 -15445.124} C_VEL
LIN {X 0,Y 319.572,Z 314.676,A -85,B 0,C 180,E1 -15449.058,E2 -15449.058} C_VEL
LIN {X 0,Y 319.599,Z 314.669,A -85,B 0,C 180,E1 -15452.905,E2 -15452.905} C_VEL
LIN {X 0,Y 319.606,Z 314.675,A -85,B 0,C 180,E1 -15455.304,E2 -15455.304} C_VEL
LIN {X 0,Y 319.559,Z 314.676,A -85,B 0,C 180,E1 -15458.369,E2 -15458.369} C_VEL
LIN {X 0,Y 318.882,Z 314.765,A -85,B 0,C 180,E1 -15459.422,E2 -15459.422} C_VEL
LIN {X 0,Y 316.03,Z 315.12,A -85,B 0,C 180,E1 -15461.135,E2 -15461.135} C_VEL
LIN {X 0,Y 313.645,Z 315.414,A -85,B 0,C 180,E1 -15462.524,E2 -15462.524} C_VEL
LIN {X 0,Y 312.657,Z 315.538,A -85,B 0,C 180,E1 -15463.599,E2 -15463.599} C_VEL
LIN {X 0,Y 312.595,Z 315.543,A -85,B 0,C 180,E1 -15463.963,E2 -15463.963} C_VEL
LIN {X 0,Y 312.639,Z 315.543,A -85,B 0,C 180,E1 -15467.009,E2 -15467.009} C_VEL
LIN {X 0,Y 312.797,Z 315.522,A -85,B 0,C 180,E1 -15471.344,E2 -15471.344} C_VEL
LIN {X 0,Y 312.898,Z 315.507,A -85,B 0,C 180,E1 -15473.552,E2 -15473.552} C_VEL
LIN {X 0,Y 312.936,Z 315.502,A -85,B 0,C 180,E1 -15477.426,E2 -15477.426} C_VEL
LIN {X 0,Y 313.087,Z 315.483,A -85,B 0,C 180,E1 -15480,E2 -15480} C_VEL
LIN {X 0,Y 312.927,Z 315.506,A -85,B 0,C 180,E1 -15482.575,E2 -15482.575} C_VEL
LIN {X 0,Y 312.853,Z 315.514,A -85,B 0,C 180,E1 -15486.449,E2 -15486.449} C_VEL
LIN {X 0,Y 312.754,Z 315.526,A -85,B 0,C 180,E1 -15489.05,E2 -15489.05} C_VEL
LIN {X 0,Y 312.639,Z 315.54,A -85,B 0,C 180,E1 -15492.991,E2 -15492.991} C_VEL
LIN {X 0,Y 312.625,Z 315.54,A -85,B 0,C 180,E1 -15495.651,E2 -15495.651} C_VEL
LIN {X 0,Y 312.563,Z 315.548,A -85,B 0,C 180,E1 -15499.711,E2 -15499.711} C_VEL
LIN {X 0,Y 312.528,Z 315.554,A -85,B 0,C 180,E1 -15502.78,E2 -15502.78} C_VEL
LIN {X 0,Y 312.541,Z 315.551,A -85,B 0,C 180,E1 -15505.911,E2 -15505.911} C_VEL
LIN {X 0,Y 312.507,Z 315.555,A -85,B 0,C 180,E1 -15509.654,E2 -15509.654} C_VEL
LIN {X 0,Y 312.523,Z 315.554,A -85,B 0,C 180,E1 -15513.689,E2 -15513.689} C_VEL
LIN {X 0,Y 312.528,Z 315.553,A -85,B 0,C 180,E1 -15517.385,E2 -15517.385} C_VEL
LIN {X 0,Y 312.492,Z 315.561,A -85,B 0,C 180,E1 -15520.709,E2 -15520.709} C_VEL
LIN {X 0,Y 312.542,Z 315.611,A -85,B 0,C 180,E1 -15523.232,E2 -15523.232} C_VEL
LIN {X 0,Y 313.536,Z 321.048,A -85,B 0,C 180,E1 -15526.76,E2 -15526.76} C_VEL
LIN {X 0,Y 314.627,Z 327.075,A -85,B 0,C 180,E1 -15530.459,E2 -15530.459} C_VEL
LIN {X 0,Y 315.186,Z 331.385,A -85,B 0,C 180,E1 -15532.983,E2 -15532.983} C_VEL
LIN {X 0,Y 314.612,Z 336.421,A -85,B 0,C 180,E1 -15535.744,E2 -15535.744} C_VEL
LIN {X 0,Y 313.524,Z 343.83,A -85,B 0,C 180,E1 -15539.711,E2 -15539.711} C_VEL
LIN {X 0,Y 312.633,Z 350.669,A -85,B 0,C 180,E1 -15543.282,E2 -15543.282} C_VEL
LIN {X 0,Y 311.835,Z 358.935,A -85,B 0,C 180,E1 -15547.525,E2 -15547.525} C_VEL
LIN {X 0,Y 311.778,Z 359.916,A -85,B 0,C 180,E1 -15547.925,E2 -15547.925} C_VEL
LIN {X 0,Y 313.759,Z 373.984,A -85,B 0,C 180,E1 -15548.654,E2 -15548.654} C_VEL
LIN {X 0,Y 315.243,Z 387.114,A -85,B 0,C 180,E1 -15549.595,E2 -15549.595} C_VEL
LIN {X 0,Y 316.141,Z 399.196,A -85,B 0,C 180,E1 -15550.69,E2 -15550.69} C_VEL
LIN {X 0,Y 316.398,Z 407.093,A -85,B 0,C 180,E1 -15551.547,E2 -15551.547} C_VEL
LIN {X 0,Y 314.953,Z 418.451,A -85,B 0,C 180,E1 -15552.97,E2 -15552.97} C_VEL
LIN {X 0,Y 313.819,Z 427.695,A -85,B 0,C 180,E1 -15554.411,E2 -15554.411} C_VEL
LIN {X 0,Y 312.893,Z 436.17,A -85,B 0,C 180,E1 -15556.027,E2 -15556.027} C_VEL
LIN {X 0,Y 311.99,Z 444.443,A -85,B 0,C 180,E1 -15557.973,E2 -15557.973} C_VEL
LIN {X 0,Y 311.49,Z 450.093,A -85,B 0,C 180,E1 -15559.601,E2 -15559.601} C_VEL
LIN {X 0,Y 311.151,Z 455.597,A -85,B 0,C 180,E1 -15561.557,E2 -15561.557} C_VEL
LIN {X 0,Y 311.032,Z 460.494,A -85,B 0,C 180,E1 -15563.836,E2 -15563.836} C_VEL
LIN {X 0,Y 310.969,Z 463.879,A -85,B 0,C 180,E1 -15566.112,E2 -15566.112} C_VEL
LIN {X 0,Y 311.105,Z 465.19,A -85,B 0,C 180,E1 -15567.41,E2 -15567.41} C_VEL
LIN {X 0,Y 311.214,Z 466.084,A -85,B 0,C 180,E1 -15568.706,E2 -15568.706} C_VEL
LIN {X 0,Y 311.218,Z 466.559,A -85,B 0,C 180,E1 -15570,E2 -15570} C_VEL
LIN {X 0,Y 311.19,Z 466.581,A -85,B 0,C 180,E1 -15571.294,E2 -15571.294} C_VEL
LIN {X 0,Y 311.024,Z 466.178,A -85,B 0,C 180,E1 -15572.59,E2 -15572.59} C_VEL
LIN {X 0,Y 310.925,Z 465.38,A -85,B 0,C 180,E1 -15573.888,E2 -15573.888} C_VEL
LIN {X 0,Y 310.841,Z 463.404,A -85,B 0,C 180,E1 -15575.829,E2 -15575.829} C_VEL
LIN {X 0,Y 310.99,Z 460.443,A -85,B 0,C 180,E1 -15577.793,E2 -15577.793} C_VEL
LIN {X 0,Y 311.302,Z 456.466,A -85,B 0,C 180,E1 -15579.748,E2 -15579.748} C_VEL
LIN {X 0,Y 311.887,Z 451.39,A -85,B 0,C 180,E1 -15581.701,E2 -15581.701} C_VEL
LIN {X 0,Y 313.173,Z 443.93,A -85,B 0,C 180,E1 -15583.96,E2 -15583.96} C_VEL
LIN {X 0,Y 314.553,Z 435.713,A -85,B 0,C 180,E1 -15585.919,E2 -15585.919} C_VEL
LIN {X 0,Y 315.821,Z 427.751,A -85,B 0,C 180,E1 -15587.483,E2 -15587.483} C_VEL
LIN {X 0,Y 317.861,Z 416.903,A -85,B 0,C 180,E1 -15589.202,E2 -15589.202} C_VEL
LIN {X 0,Y 319.083,Z 408.541,A -85,B 0,C 180,E1 -15590.298,E2 -15590.298} C_VEL
LIN {X 0,Y 319.282,Z 397.063,A -85,B 0,C 180,E1 -15591.659,E2 -15591.659} C_VEL
LIN {X 0,Y 318.51,Z 385.115,A -85,B 0,C 180,E1 -15592.876,E2 -15592.876} C_VEL
LIN {X 0,Y 316.742,Z 373.125,A -85,B 0,C 180,E1 -15593.952,E2 -15593.952} C_VEL
LIN {X 0,Y 313.443,Z 358.973,A -85,B 0,C 180,E1 -15595.09,E2 -15595.09} C_VEL
LIN {X 0,Y 312.478,Z 355.236,A -85,B 0,C 180,E1 -15595.379,E2 -15595.379} C_VEL
LIN {X 0,Y 313.368,Z 348.507,A -85,B 0,C 180,E1 -15598.994,E2 -15598.994} C_VEL
LIN {X 0,Y 314.542,Z 341.088,A -85,B 0,C 180,E1 -15603.19,E2 -15603.19} C_VEL
LIN {X 0,Y 315.79,Z 334.851,A -85,B 0,C 180,E1 -15606.934,E2 -15606.934} C_VEL
LIN {X 0,Y 315.365,Z 331.149,A -85,B 0,C 180,E1 -15609.459,E2 -15609.459} C_VEL
LIN {X 0,Y 314.684,Z 327.074,A -85,B 0,C 180,E1 -15612.523,E2 -15612.523} C_VEL
LIN {X 0,Y 313.886,Z 322.883,A -85,B 0,C 180,E1 -15616.044,E2 -15616.044} C_VEL
LIN {X 0,Y 313.214,Z 319.132,A -85,B 0,C 180,E1 -15619.722,E2 -15619.722} C_VEL
LIN {X 0,Y 312.591,Z 315.885,A -85,B 0,C 180,E1 -15623.402,E2 -15623.402} C_VEL
LIN {X 0,Y 312.536,Z 315.557,A -85,B 0,C 180,E1 -15624.221,E2 -15624.221} C_VEL
LIN {X 0,Y 312.508,Z 315.559,A -85,B 0,C 180,E1 -15627.334,E2 -15627.334} C_VEL
LIN {X 0,Y 312.556,Z 315.553,A -85,B 0,C 180,E1 -15631.276,E2 -15631.276} C_VEL
LIN {X 0,Y 312.589,Z 315.549,A -85,B 0,C 180,E1 -15634.711,E2 -15634.711} C_VEL
LIN {X 0,Y 312.591,Z 315.545,A -85,B 0,C 180,E1 -15637.529,E2 -15637.529} C_VEL
LIN {X 0,Y 312.643,Z 315.54,A -85,B 0,C 180,E1 -15641.656,E2 -15641.656} C_VEL
LIN {X 0,Y 312.698,Z 315.536,A -85,B 0,C 180,E1 -15645.686,E2 -15645.686} C_VEL
LIN {X 0,Y 312.69,Z 315.535,A -85,B 0,C 180,E1 -15649.641,E2 -15649.641} C_VEL
LIN {X 0,Y 312.821,Z 315.521,A -85,B 0,C 180,E1 -15652.253,E2 -15652.253} C_VEL
LIN {X 0,Y 312.709,Z 315.533,A -85,B 0,C 180,E1 -15654.842,E2 -15654.842} C_VEL
LIN {X 0,Y 312.993,Z 315.497,A -85,B 0,C 180,E1 -15658.713,E2 -15658.713} C_VEL
LIN {X 0,Y 312.993,Z 315.499,A -85,B 0,C 180,E1 -15661.286,E2 -15661.286} C_VEL
LIN {X 0,Y 312.697,Z 315.536,A -85,B 0,C 180,E1 -15663.866,E2 -15663.866} C_VEL
LIN {X 0,Y 312.715,Z 315.609,A -85,B 0,C 180,E1 -15665.157,E2 -15665.157} C_VEL
LIN {X 0,Y 313.027,Z 317.033,A -85,B 0,C 180,E1 -15667.742,E2 -15667.742} C_VEL
LIN {X 0,Y 312.82,Z 319.498,A -85,B 0,C 180,E1 -15671.665,E2 -15671.665} C_VEL
LIN {X 0,Y 312.769,Z 320.261,A -85,B 0,C 180,E1 -15672.82,E2 -15672.82} C_VEL
LIN {X 0,Y 314.028,Z 323.512,A -85,B 0,C 180,E1 -15673.138,E2 -15673.138} C_VEL
LIN {X 0,Y 318.553,Z 334.493,A -85,B 0,C 180,E1 -15674.327,E2 -15674.327} C_VEL
LIN {X 0,Y 321.884,Z 344.942,A -85,B 0,C 180,E1 -15675.513,E2 -15675.513} C_VEL
LIN {X 0,Y 323.726,Z 353.597,A -85,B 0,C 180,E1 -15676.553,E2 -15676.553} C_VEL
LIN {X 0,Y 322.13,Z 365.147,A -85,B 0,C 180,E1 -15677.785,E2 -15677.785} C_VEL
LIN {X 0,Y 320.476,Z 375.6,A -85,B 0,C 180,E1 -15679.205,E2 -15679.205} C_VEL
LIN {X 0,Y 318.593,Z 386.065,A -85,B 0,C 180,E1 -15680.978,E2 -15680.978} C_VEL
LIN {X 0,Y 316.907,Z 394.747,A -85,B 0,C 180,E1 -15682.836,E2 -15682.836} C_VEL
LIN {X 0,Y 315.59,Z 401.217,A -85,B 0,C 180,E1 -15684.549,E2 -15684.549} C_VEL
LIN {X 0,Y 314.283,Z 407.322,A -85,B 0,C 180,E1 -15686.567,E2 -15686.567} C_VEL
LIN {X 0,Y 313.133,Z 412.737,A -85,B 0,C 180,E1 -15688.916,E2 -15688.916} C_VEL
LIN {X 0,Y 312.241,Z 416.447,A -85,B 0,C 180,E1 -15691.205,E2 -15691.205} C_VEL
LIN {X 0,Y 311.588,Z 418.771,A -85,B 0,C 180,E1 -15693.43,E2 -15693.43} C_VEL
LIN {X 0,Y 311.146,Z 419.983,A -85,B 0,C 180,E1 -15695.964,E2 -15695.964} C_VEL
LIN {X 0,Y 311.018,Z 419.883,A -85,B 0,C 180,E1 -15697.731,E2 -15697.731} C_VEL
LIN {X 0,Y 311.04,Z 418.841,A -85,B 0,C 180,E1 -15699.804,E2 -15699.804} C_VEL
LIN {X 0,Y 311.239,Z 416.817,A -85,B 0,C 180,E1 -15701.826,E2 -15701.826} C_VEL
LIN {X 0,Y 311.704,Z 412.842,A -85,B 0,C 180,E1 -15704.343,E2 -15704.343} C_VEL
LIN {X 0,Y 312.118,Z 409.036,A -85,B 0,C 180,E1 -15706.1,E2 -15706.1} C_VEL
LIN {X 0,Y 312.793,Z 403.264,A -85,B 0,C 180,E1 -15708.17,E2 -15708.17} C_VEL
LIN {X 0,Y 313.572,Z 396.609,A -85,B 0,C 180,E1 -15710.071,E2 -15710.071} C_VEL
LIN {X 0,Y 314.539,Z 388.821,A -85,B 0,C 180,E1 -15711.875,E2 -15711.875} C_VEL
LIN {X 0,Y 315.659,Z 379.683,A -85,B 0,C 180,E1 -15713.596,E2 -15713.596} C_VEL
LIN {X 0,Y 316.882,Z 369.445,A -85,B 0,C 180,E1 -15715.145,E2 -15715.145} C_VEL
LIN {X 0,Y 317.924,Z 358.845,A -85,B 0,C 180,E1 -15716.451,E2 -15716.451} C_VEL
LIN {X 0,Y 318.93,Z 347.799,A -85,B 0,C 180,E1 -15717.54,E2 -15717.54} C_VEL
LIN {X 0,Y 318.697,Z 344.288,A -85,B 0,C 180,E1 -15717.858,E2 -15717.858} C_VEL
LIN {X 0,Y 316.029,Z 332.318,A -85,B 0,C 180,E1 -15718.904,E2 -15718.904} C_VEL
LIN {X 0,Y 312.772,Z 319.749,A -85,B 0,C 180,E1 -15719.77,E2 -15719.77} C_VEL
LIN {X 0,Y 311.688,Z 315.661,A -85,B 0,C 180,E1 -15720.027,E2 -15720.027} C_VEL
LIN {X 0,Y 312.209,Z 315.592,A -85,B 0,C 180,E1 -15724.213,E2 -15724.213} C_VEL
LIN {X 0,Y 312.479,Z 315.561,A -85,B 0,C 180,E1 -15727.521,E2 -15727.521} C_VEL
LIN {X 0,Y 312.567,Z 315.549,A -85,B 0,C 180,E1 -15731.652,E2 -15731.652} C_VEL
LIN {X 0,Y 312.686,Z 315.533,A -85,B 0,C 180,E1 -15735.686,E2 -15735.686} C_VEL
LIN {X 0,Y 312.699,Z 315.532,A -85,B 0,C 180,E1 -15739.642,E2 -15739.642} C_VEL
LIN {X 0,Y 312.803,Z 315.519,A -85,B 0,C 180,E1 -15742.252,E2 -15742.252} C_VEL
LIN {X 0,Y 312.707,Z 315.535,A -85,B 0,C 180,E1 -15744.842,E2 -15744.842} C_VEL
LIN {X 0,Y 312.991,Z 315.499,A -85,B 0,C 180,E1 -15748.713,E2 -15748.713} C_VEL
LIN {X 0,Y 312.99,Z 315.495,A -85,B 0,C 180,E1 -15751.287,E2 -15751.287} C_VEL
LIN {X 0,Y 312.693,Z 315.532,A -85,B 0,C 180,E1 -15753.866,E2 -15753.866} C_VEL
LIN {X 0,Y 312.85,Z 315.516,A -85,B 0,C 180,E1 -15756.449,E2 -15756.449} C_VEL
LIN {X 0,Y 312.756,Z 315.525,A -85,B 0,C 180,E1 -15759.05,E2 -15759.05} C_VEL
LIN {X 0,Y 312.635,Z 315.54,A -85,B 0,C 180,E1 -15762.991,E2 -15762.991} C_VEL
LIN {X 0,Y 312.639,Z 315.538,A -85,B 0,C 180,E1 -15765.65,E2 -15765.65} C_VEL
LIN {X 0,Y 312.631,Z 315.539,A -85,B 0,C 180,E1 -15769.237,E2 -15769.237} C_VEL
LIN {X 0,Y 312.547,Z 315.551,A -85,B 0,C 180,E1 -15772.789,E2 -15772.789} C_VEL
LIN {X 0,Y 312.604,Z 315.546,A -85,B 0,C 180,E1 -15775.936,E2 -15775.936} C_VEL
LIN {X 0,Y 312.546,Z 315.551,A -85,B 0,C 180,E1 -15779.65,E2 -15779.65} C_VEL
LIN {X 0,Y 312.52,Z 315.555,A -85,B 0,C 180,E1 -15783.689,E2 -15783.689} C_VEL
LIN {X 0,Y 312.538,Z 315.552,A -85,B 0,C 180,E1 -15787.384,E2 -15787.384} C_VEL
LIN {X 0,Y 312.491,Z 315.557,A -85,B 0,C 180,E1 -15790.709,E2 -15790.709} C_VEL
LIN {X 0,Y 312.453,Z 315.564,A -85,B 0,C 180,E1 -15794.21,E2 -15794.21} C_VEL
LIN {X 0,Y 312.486,Z 315.561,A -85,B 0,C 180,E1 -15797.919,E2 -15797.919} C_VEL
LIN {X 0,Y 312.537,Z 315.554,A -85,B 0,C 180,E1 -15801.911,E2 -15801.911} C_VEL
LIN {X 0,Y 312.508,Z 315.558,A -85,B 0,C 180,E1 -15805.79,E2 -15805.79} C_VEL
LIN {X 0,Y 312.526,Z 315.553,A -85,B 0,C 180,E1 -15808.854,E2 -15808.854} C_VEL
LIN {X 0,Y 312.577,Z 315.548,A -85,B 0,C 180,E1 -15811.825,E2 -15811.825} C_VEL
LIN {X 0,Y 312.587,Z 315.545,A -85,B 0,C 180,E1 -15814.711,E2 -15814.711} C_VEL
LIN {X 0,Y 312.523,Z 315.553,A -85,B 0,C 180,E1 -15818.367,E2 -15818.367} C_VEL
LIN {X 0,Y 312.585,Z 315.547,A -85,B 0,C 180,E1 -15821.653,E2 -15821.653} C_VEL
LIN {X 0,Y 312.595,Z 315.543,A -85,B 0,C 180,E1 -15823.963,E2 -15823.963} C_VEL
LIN {X 0,Y 311.979,Z 315.625,A -85,B 0,C 180,E1 -15825.038,E2 -15825.038} C_VEL
LIN {X 0,Y 309.152,Z 315.978,A -85,B 0,C 180,E1 -15826.788,E2 -15826.788} C_VEL
LIN {X 0,Y 306.733,Z 316.279,A -85,B 0,C 180,E1 -15828.208,E2 -15828.208} C_VEL
LIN {X 0,Y 305.705,Z 316.405,A -85,B 0,C 180,E1 -15829.307,E2 -15829.307} C_VEL
LIN {X 0,Y 305.629,Z 316.412,A -85,B 0,C 180,E1 -15829.68,E2 -15829.68} C_VEL
LIN {X 0,Y 305.838,Z 316.388,A -85,B 0,C 180,E1 -15833.402,E2 -15833.402} C_VEL
LIN {X 0,Y 305.885,Z 316.381,A -85,B 0,C 180,E1 -15837.366,E2 -15837.366} C_VEL
LIN {X 0,Y 306.042,Z 316.36,A -85,B 0,C 180,E1 -15840,E2 -15840} C_VEL
LIN {X 0,Y 305.876,Z 316.385,A -85,B 0,C 180,E1 -15842.634,E2 -15842.634} C_VEL
LIN {X 0,Y 305.797,Z 316.394,A -85,B 0,C 180,E1 -15846.599,E2 -15846.599} C_VEL
LIN {X 0,Y 305.697,Z 316.404,A -85,B 0,C 180,E1 -15849.261,E2 -15849.261} C_VEL
LIN {X 0,Y 305.591,Z 316.416,A -85,B 0,C 180,E1 -15853.296,E2 -15853.296} C_VEL
LIN {X 0,Y 305.555,Z 316.422,A -85,B 0,C 180,E1 -15856.022,E2 -15856.022} C_VEL
LIN {X 0,Y 305.545,Z 316.422,A -85,B 0,C 180,E1 -15859.426,E2 -15859.426} C_VEL
LIN {X 0,Y 305.489,Z 316.429,A -85,B 0,C 180,E1 -15863.039,E2 -15863.039} C_VEL
LIN {X 0,Y 305.481,Z 316.432,A -85,B 0,C 180,E1 -15866.2,E2 -15866.2} C_VEL
LIN {X 0,Y 305.466,Z 316.431,A -85,B 0,C 180,E1 -15869.039,E2 -15869.039} C_VEL
LIN {X 0,Y 305.44,Z 316.438,A -85,B 0,C 180,E1 -15871.953,E2 -15871.953} C_VEL
LIN {X 0,Y 305.465,Z 316.432,A -85,B 0,C 180,E1 -15875.113,E2 -15875.113} C_VEL
LIN {X 0,Y 305.469,Z 316.434,A -85,B 0,C 180,E1 -15878.533,E2 -15878.533} C_VEL
LIN {X 0,Y 305.485,Z 316.433,A -85,B 0,C 180,E1 -15882.874,E2 -15882.874} C_VEL
LIN {X 0,Y 306.501,Z 321.936,A -85,B 0,C 180,E1 -15886.536,E2 -15886.536} C_VEL
LIN {X 0,Y 307.555,Z 327.761,A -85,B 0,C 180,E1 -15890.22,E2 -15890.22} C_VEL
LIN {X 0,Y 308.161,Z 332.334,A -85,B 0,C 180,E1 -15892.961,E2 -15892.961} C_VEL
LIN {X 0,Y 307.46,Z 337.761,A -85,B 0,C 180,E1 -15896.009,E2 -15896.009} C_VEL
LIN {X 0,Y 306.461,Z 344.524,A -85,B 0,C 180,E1 -15899.7,E2 -15899.7} C_VEL
LIN {X 0,Y 305.441,Z 352.199,A -85,B 0,C 180,E1 -15903.815,E2 -15903.815} C_VEL
LIN {X 0,Y 304.746,Z 359.2,A -85,B 0,C 180,E1 -15907.502,E2 -15907.502} C_VEL
LIN {X 0,Y 306.75,Z 373.472,A -85,B 0,C 180,E1 -15908.267,E2 -15908.267} C_VEL
LIN {X 0,Y 308.182,Z 386.549,A -85,B 0,C 180,E1 -15909.228,E2 -15909.228} C_VEL
LIN {X 0,Y 309.132,Z 399.179,A -85,B 0,C 180,E1 -15910.407,E2 -15910.407} C_VEL
LIN {X 0,Y 309.42,Z 406.994,A -85,B 0,C 180,E1 -15911.287,E2 -15911.287} C_VEL
LIN {X 0,Y 307.97,Z 418.278,A -85,B 0,C 180,E1 -15912.742,E2 -15912.742} C_VEL
LIN {X 0,Y 306.587,Z 428.883,A -85,B 0,C 180,E1 -15914.479,E2 -15914.479} C_VEL
LIN {X 0,Y 305.749,Z 436.612,A -85,B 0,C 180,E1 -15916.033,E2 -15916.033} C_VEL
LIN {X 0,Y 304.849,Z 444.719,A -85,B 0,C 180,E1 -15918.025,E2 -15918.025} C_VEL
LIN {X 0,Y 304.297,Z 451.234,A -85,B 0,C 180,E1 -15920.025,E2 -15920.025} C_VEL
LIN {X 0,Y 304.005,Z 456.38,A -85,B 0,C 180,E1 -15922.027,E2 -15922.027} C_VEL
LIN {X 0,Y 303.947,Z 460.063,A -85,B 0,C 180,E1 -15923.863,E2 -15923.863} C_VEL
LIN {X 0,Y 303.897,Z 463.215,A -85,B 0,C 180,E1 -15926.022,E2 -15926.022} C_VEL
LIN {X 0,Y 304.012,Z 464.553,A -85,B 0,C 180,E1 -15927.35,E2 -15927.35} C_VEL
LIN {X 0,Y 304.152,Z 465.475,A -85,B 0,C 180,E1 -15928.676,E2 -15928.676} C_VEL
LIN {X 0,Y 304.158,Z 465.977,A -85,B 0,C 180,E1 -15930,E2 -15930} C_VEL
LIN {X 0,Y 304.126,Z 466.047,A -85,B 0,C 180,E1 -15931.324,E2 -15931.324} C_VEL
LIN {X 0,Y 303.847,Z 464.89,A -85,B 0,C 180,E1 -15933.979,E2 -15933.979} C_VEL
LIN {X 0,Y 303.747,Z 463.193,A -85,B 0,C 180,E1 -15935.774,E2 -15935.774} C_VEL
LIN {X 0,Y 303.925,Z 460.059,A -85,B 0,C 180,E1 -15937.975,E2 -15937.975} C_VEL
LIN {X 0,Y 304.277,Z 456.156,A -85,B 0,C 180,E1 -15939.976,E2 -15939.976} C_VEL
LIN {X 0,Y 304.9,Z 451.152,A -85,B 0,C 180,E1 -15941.973,E2 -15941.973} C_VEL
LIN {X 0,Y 306.248,Z 443.766,A -85,B 0,C 180,E1 -15944.282,E2 -15944.282} C_VEL
LIN {X 0,Y 307.606,Z 436.263,A -85,B 0,C 180,E1 -15946.153,E2 -15946.153} C_VEL
LIN {X 0,Y 309.051,Z 427.816,A -85,B 0,C 180,E1 -15947.879,E2 -15947.879} C_VEL
LIN {X 0,Y 311.176,Z 417.15,A -85,B 0,C 180,E1 -15949.631,E2 -15949.631} C_VEL
LIN {X 0,Y 312.427,Z 409.005,A -85,B 0,C 180,E1 -15950.75,E2 -15950.75} C_VEL
LIN {X 0,Y 312.709,Z 397.884,A -85,B 0,C 180,E1 -15952.127,E2 -15952.127} C_VEL
LIN {X 0,Y 311.984,Z 385.736,A -85,B 0,C 180,E1 -15953.434,E2 -15953.434} C_VEL
LIN {X 0,Y 310.187,Z 373.378,A -85,B 0,C 180,E1 -15954.61,E2 -15954.61} C_VEL
LIN {X 0,Y 307.319,Z 361.239,A -85,B 0,C 180,E1 -15955.669,E2 -15955.669} C_VEL
LIN {X 0,Y 305.616,Z 354.594,A -85,B 0,C 180,E1 -15956.186,E2 -15956.186} C_VEL
LIN {X 0,Y 306.633,Z 347.276,A -85,B 0,C 180,E1 -15960.281,E2 -15960.281} C_VEL
LIN {X 0,Y 308.084,Z 339.637,A -85,B 0,C 180,E1 -15964.791,E2 -15964.791} C_VEL
LIN {X 0,Y 308.806,Z 335.813,A -85,B 0,C 180,E1 -15967.197,E2 -15967.197} C_VEL
LIN {X 0,Y 308.226,Z 331.342,A -85,B 0,C 180,E1 -15970.402,E2 -15970.402} C_VEL
LIN {X 0,Y 307.561,Z 327.701,A -85,B 0,C 180,E1 -15973.277,E2 -15973.277} C_VEL
LIN {X 0,Y 306.837,Z 323.911,A -85,B 0,C 180,E1 -15976.596,E2 -15976.596} C_VEL
LIN {X 0,Y 306.265,Z 320.538,A -85,B 0,C 180,E1 -15980.019,E2 -15980.019} C_VEL
LIN {X 0,Y 305.723,Z 317.542,A -85,B 0,C 180,E1 -15983.571,E2 -15983.571} C_VEL
LIN {X 0,Y 305.465,Z 316.433,A -85,B 0,C 180,E1 -15985.176,E2 -15985.176} C_VEL
LIN {X 0,Y 305.467,Z 316.435,A -85,B 0,C 180,E1 -15989.591,E2 -15989.591} C_VEL
LIN {X 0,Y 305.525,Z 316.428,A -85,B 0,C 180,E1 -15992.609,E2 -15992.609} C_VEL
LIN {X 0,Y 305.512,Z 316.426,A -85,B 0,C 180,E1 -15995.539,E2 -15995.539} C_VEL
LIN {X 0,Y 305.525,Z 316.425,A -85,B 0,C 180,E1 -15999.815,E2 -15999.815} C_VEL
LIN {X 0,Y 305.579,Z 316.419,A -85,B 0,C 180,E1 -16002.603,E2 -16002.603} C_VEL
LIN {X 0,Y 305.653,Z 316.412,A -85,B 0,C 180,E1 -16005.349,E2 -16005.349} C_VEL
LIN {X 0,Y 305.628,Z 316.413,A -85,B 0,C 180,E1 -16009.399,E2 -16009.399} C_VEL
LIN {X 0,Y 305.768,Z 316.398,A -85,B 0,C 180,E1 -16012.073,E2 -16012.073} C_VEL
LIN {X 0,Y 305.678,Z 316.409,A -85,B 0,C 180,E1 -16014.723,E2 -16014.723} C_VEL
LIN {X 0,Y 305.96,Z 316.373,A -85,B 0,C 180,E1 -16018.684,E2 -16018.684} C_VEL
LIN {X 0,Y 305.96,Z 316.375,A -85,B 0,C 180,E1 -16021.316,E2 -16021.316} C_VEL
LIN {X 0,Y 305.647,Z 316.414,A -85,B 0,C 180,E1 -16023.955,E2 -16023.955} C_VEL
LIN {X 0,Y 305.992,Z 317.717,A -85,B 0,C 180,E1 -16026.594,E2 -16026.594} C_VEL
LIN {X 0,Y 305.969,Z 319.262,A -85,B 0,C 180,E1 -16029.252,E2 -16029.252} C_VEL
LIN {X 0,Y 305.819,Z 320.967,A -85,B 0,C 180,E1 -16031.978,E2 -16031.978} C_VEL
LIN {X 0,Y 306.993,Z 324.046,A -85,B 0,C 180,E1 -16032.309,E2 -16032.309} C_VEL
LIN {X 0,Y 311.142,Z 333.396,A -85,B 0,C 180,E1 -16033.386,E2 -16033.386} C_VEL
LIN {X 0,Y 314.977,Z 344.865,A -85,B 0,C 180,E1 -16034.757,E2 -16034.757} C_VEL
LIN {X 0,Y 317.269,Z 354.607,A -85,B 0,C 180,E1 -16035.992,E2 -16035.992} C_VEL
LIN {X 0,Y 315.893,Z 365.161,A -85,B 0,C 180,E1 -16037.153,E2 -16037.153} C_VEL
LIN {X 0,Y 314.154,Z 375.676,A -85,B 0,C 180,E1 -16038.585,E2 -16038.585} C_VEL
LIN {X 0,Y 312.49,Z 384.451,A -85,B 0,C 180,E1 -16040.058,E2 -16040.058} C_VEL
LIN {X 0,Y 310.616,Z 393.463,A -85,B 0,C 180,E1 -16041.925,E2 -16041.925} C_VEL
LIN {X 0,Y 309.077,Z 400.724,A -85,B 0,C 180,E1 -16043.804,E2 -16043.804} C_VEL
LIN {X 0,Y 307.777,Z 406.639,A -85,B 0,C 180,E1 -16045.713,E2 -16045.713} C_VEL
LIN {X 0,Y 306.459,Z 412.212,A -85,B 0,C 180,E1 -16048.042,E2 -16048.042} C_VEL
LIN {X 0,Y 305.458,Z 416.328,A -85,B 0,C 180,E1 -16050.409,E2 -16050.409} C_VEL
LIN {X 0,Y 304.913,Z 418.281,A -85,B 0,C 180,E1 -16052.014,E2 -16052.014} C_VEL
LIN {X 0,Y 304.447,Z 419.762,A -85,B 0,C 180,E1 -16053.793,E2 -16053.793} C_VEL
LIN {X 0,Y 304.08,Z 420.557,A -85,B 0,C 180,E1 -16056.007,E2 -16056.007} C_VEL
LIN {X 0,Y 303.905,Z 420.061,A -85,B 0,C 180,E1 -16058.637,E2 -16058.637} C_VEL
LIN {X 0,Y 303.996,Z 418.904,A -85,B 0,C 180,E1 -16060.34,E2 -16060.34} C_VEL
LIN {X 0,Y 304.233,Z 416.688,A -85,B 0,C 180,E1 -16062.334,E2 -16062.334} C_VEL
LIN {X 0,Y 304.614,Z 413.468,A -85,B 0,C 180,E1 -16064.338,E2 -16064.338} C_VEL
LIN {X 0,Y 305.223,Z 408,A -85,B 0,C 180,E1 -16066.804,E2 -16066.804} C_VEL
LIN {X 0,Y 305.871,Z 402.606,A -85,B 0,C 180,E1 -16068.677,E2 -16068.677} C_VEL
LIN {X 0,Y 306.778,Z 395.621,A -85,B 0,C 180,E1 -16070.634,E2 -16070.634} C_VEL
LIN {X 0,Y 307.772,Z 387.456,A -85,B 0,C 180,E1 -16072.478,E2 -16072.478} C_VEL
LIN {X 0,Y 309.07,Z 377.313,A -85,B 0,C 180,E1 -16074.322,E2 -16074.322} C_VEL
LIN {X 0,Y 310.285,Z 367.093,A -85,B 0,C 180,E1 -16075.819,E2 -16075.819} C_VEL
LIN {X 0,Y 311.449,Z 355.174,A -85,B 0,C 180,E1 -16077.209,E2 -16077.209} C_VEL
LIN {X 0,Y 312.083,Z 348.462,A -85,B 0,C 180,E1 -16077.857,E2 -16077.857} C_VEL
LIN {X 0,Y 311.42,Z 343.347,A -85,B 0,C 180,E1 -16078.352,E2 -16078.352} C_VEL
LIN {X 0,Y 308.382,Z 330.208,A -85,B 0,C 180,E1 -16079.483,E2 -16079.483} C_VEL
LIN {X 0,Y 305.065,Z 318.141,A -85,B 0,C 180,E1 -16080.309,E2 -16080.309} C_VEL
LIN {X 0,Y 304.689,Z 316.531,A -85,B 0,C 180,E1 -16080.412,E2 -16080.412} C_VEL
LIN {X 0,Y 305.146,Z 316.473,A -85,B 0,C 180,E1 -16084.049,E2 -16084.049} C_VEL
LIN {X 0,Y 305.373,Z 316.447,A -85,B 0,C 180,E1 -16087.011,E2 -16087.011} C_VEL
LIN {X 0,Y 305.517,Z 316.431,A -85,B 0,C 180,E1 -16091.213,E2 -16091.213} C_VEL
LIN {X 0,Y 305.627,Z 316.415,A -85,B 0,C 180,E1 -16095.348,E2 -16095.348} C_VEL
LIN {X 0,Y 305.636,Z 316.413,A -85,B 0,C 180,E1 -16099.4,E2 -16099.4} C_VEL
LIN {X 0,Y 305.752,Z 316.397,A -85,B 0,C 180,E1 -16102.073,E2 -16102.073} C_VEL
LIN {X 0,Y 305.676,Z 316.41,A -85,B 0,C 180,E1 -16104.723,E2 -16104.723} C_VEL
LIN {X 0,Y 305.958,Z 316.375,A -85,B 0,C 180,E1 -16108.684,E2 -16108.684} C_VEL
LIN {X 0,Y 305.957,Z 316.371,A -85,B 0,C 180,E1 -16111.316,E2 -16111.316} C_VEL
LIN {X 0,Y 305.676,Z 316.407,A -85,B 0,C 180,E1 -16115.277,E2 -16115.277} C_VEL
LIN {X 0,Y 305.752,Z 316.397,A -85,B 0,C 180,E1 -16117.927,E2 -16117.927} C_VEL
LIN {X 0,Y 305.604,Z 316.416,A -85,B 0,C 180,E1 -16121.945,E2 -16121.945} C_VEL
LIN {X 0,Y 305.639,Z 316.411,A -85,B 0,C 180,E1 -16125.035,E2 -16125.035} C_VEL
LIN {X 0,Y 305.577,Z 316.418,A -85,B 0,C 180,E1 -16129.445,E2 -16129.445} C_VEL
LIN {X 0,Y 305.491,Z 316.429,A -85,B 0,C 180,E1 -16133.042,E2 -16133.042} C_VEL
LIN {X 0,Y 305.549,Z 316.427,A -85,B 0,C 180,E1 -16136.227,E2 -16136.227} C_VEL
LIN {X 0,Y 305.496,Z 316.428,A -85,B 0,C 180,E1 -16139.05,E2 -16139.05} C_VEL
LIN {X 0,Y 305.445,Z 316.438,A -85,B 0,C 180,E1 -16141.952,E2 -16141.952} C_VEL
LIN {X 0,Y 305.463,Z 316.432,A -85,B 0,C 180,E1 -16145.113,E2 -16145.113} C_VEL
LIN {X 0,Y 305.468,Z 316.432,A -85,B 0,C 180,E1 -16148.533,E2 -16148.533} C_VEL
LIN {X 0,Y 305.456,Z 316.434,A -85,B 0,C 180,E1 -16152.586,E2 -16152.586} C_VEL
LIN {X 0,Y 305.427,Z 316.437,A -85,B 0,C 180,E1 -16156.345,E2 -16156.345} C_VEL
LIN {X 0,Y 305.46,Z 316.437,A -85,B 0,C 180,E1 -16159.893,E2 -16159.893} C_VEL
LIN {X 0,Y 305.483,Z 316.435,A -85,B 0,C 180,E1 -16163.632,E2 -16163.632} C_VEL
LIN {X 0,Y 305.467,Z 316.432,A -85,B 0,C 180,E1 -16166.484,E2 -16166.484} C_VEL
LIN {X 0,Y 305.498,Z 316.429,A -85,B 0,C 180,E1 -16170.95,E2 -16170.95} C_VEL
LIN {X 0,Y 305.575,Z 316.419,A -85,B 0,C 180,E1 -16174.088,E2 -16174.088} C_VEL
LIN {X 0,Y 305.478,Z 316.43,A -85,B 0,C 180,E1 -16178.401,E2 -16178.401} C_VEL
LIN {X 0,Y 305.546,Z 316.427,A -85,B 0,C 180,E1 -16181.215,E2 -16181.215} C_VEL
LIN {X 0,Y 305.629,Z 316.415,A -85,B 0,C 180,E1 -16185.348,E2 -16185.348} C_VEL
LIN {X 0,Y 305.629,Z 316.412,A -85,B 0,C 180,E1 -16189.68,E2 -16189.68} C_VEL
LIN {X 0,Y 304.983,Z 316.495,A -85,B 0,C 180,E1 -16190.781,E2 -16190.781} C_VEL
LIN {X 0,Y 302.15,Z 316.847,A -85,B 0,C 180,E1 -16192.576,E2 -16192.576} C_VEL
LIN {X 0,Y 299.73,Z 317.146,A -85,B 0,C 180,E1 -16194.031,E2 -16194.031} C_VEL
LIN {X 0,Y 298.684,Z 317.28,A -85,B 0,C 180,E1 -16195.158,E2 -16195.158} C_VEL
LIN {X 0,Y 298.595,Z 317.286,A -85,B 0,C 180,E1 -16195.54,E2 -16195.54} C_VEL
LIN {X 0,Y 298.924,Z 317.249,A -85,B 0,C 180,E1 -16198.653,E2 -16198.653} C_VEL
LIN {X 0,Y 298.924,Z 317.248,A -85,B 0,C 180,E1 -16201.347,E2 -16201.347} C_VEL
LIN {X 0,Y 298.745,Z 317.274,A -85,B 0,C 180,E1 -16206.755,E2 -16206.755} C_VEL
LIN {X 0,Y 298.629,Z 317.284,A -85,B 0,C 180,E1 -16209.482,E2 -16209.482} C_VEL
LIN {X 0,Y 298.549,Z 317.293,A -85,B 0,C 180,E1 -16213.616,E2 -16213.616} C_VEL
LIN {X 0,Y 298.49,Z 317.305,A -85,B 0,C 180,E1 -16216.412,E2 -16216.412} C_VEL
LIN {X 0,Y 298.486,Z 317.302,A -85,B 0,C 180,E1 -16219.639,E2 -16219.639} C_VEL
LIN {X 0,Y 298.427,Z 317.308,A -85,B 0,C 180,E1 -16223.6,E2 -16223.6} C_VEL
LIN {X 0,Y 298.42,Z 317.31,A -85,B 0,C 180,E1 -16226.581,E2 -16226.581} C_VEL
LIN {X 0,Y 298.403,Z 317.311,A -85,B 0,C 180,E1 -16229.643,E2 -16229.643} C_VEL
LIN {X 0,Y 298.396,Z 317.314,A -85,B 0,C 180,E1 -16232.8,E2 -16232.8} C_VEL
LIN {X 0,Y 298.449,Z 317.307,A -85,B 0,C 180,E1 -16236.808,E2 -16236.808} C_VEL
LIN {X 0,Y 298.411,Z 317.312,A -85,B 0,C 180,E1 -16239.486,E2 -16239.486} C_VEL
LIN {X 0,Y 298.459,Z 317.368,A -85,B 0,C 180,E1 -16242.609,E2 -16242.609} C_VEL
LIN {X 0,Y 299.531,Z 323.338,A -85,B 0,C 180,E1 -16246.666,E2 -16246.666} C_VEL
LIN {X 0,Y 300.733,Z 329.89,A -85,B 0,C 180,E1 -16250.877,E2 -16250.877} C_VEL
LIN {X 0,Y 301.066,Z 334.192,A -85,B 0,C 180,E1 -16253.468,E2 -16253.468} C_VEL
LIN {X 0,Y 300.18,Z 339.692,A -85,B 0,C 180,E1 -16256.619,E2 -16256.619} C_VEL
LIN {X 0,Y 299.174,Z 346.54,A -85,B 0,C 180,E1 -16260.441,E2 -16260.441} C_VEL
LIN {X 0,Y 298.279,Z 353.383,A -85,B 0,C 180,E1 -16264.198,E2 -16264.198} C_VEL
LIN {X 0,Y 297.742,Z 358.674,A -85,B 0,C 180,E1 -16267.054,E2 -16267.054} C_VEL
LIN {X 0,Y 299.747,Z 373.211,A -85,B 0,C 180,E1 -16267.876,E2 -16267.876} C_VEL
LIN {X 0,Y 301.244,Z 387.097,A -85,B 0,C 180,E1 -16268.939,E2 -16268.939} C_VEL
LIN {X 0,Y 302.115,Z 399.15,A -85,B 0,C 180,E1 -16270.11,E2 -16270.11} C_VEL
LIN {X 0,Y 302.3,Z 408.292,A -85,B 0,C 180,E1 -16271.181,E2 -16271.181} C_VEL
LIN {X 0,Y 300.884,Z 419.182,A -85,B 0,C 180,E1 -16272.674,E2 -16272.674} C_VEL
LIN {X 0,Y 299.552,Z 428.738,A -85,B 0,C 180,E1 -16274.302,E2 -16274.302} C_VEL
LIN {X 0,Y 298.826,Z 435.567,A -85,B 0,C 180,E1 -16275.703,E2 -16275.703} C_VEL
LIN {X 0,Y 297.876,Z 443.761,A -85,B 0,C 180,E1 -16277.74,E2 -16277.74} C_VEL
LIN {X 0,Y 297.277,Z 450.358,A -85,B 0,C 180,E1 -16279.787,E2 -16279.787} C_VEL
LIN {X 0,Y 296.944,Z 455.587,A -85,B 0,C 180,E1 -16281.836,E2 -16281.836} C_VEL
LIN {X 0,Y 296.882,Z 459.568,A -85,B 0,C 180,E1 -16283.857,E2 -16283.857} C_VEL
LIN {X 0,Y 296.827,Z 462.538,A -85,B 0,C 180,E1 -16285.927,E2 -16285.927} C_VEL
LIN {X 0,Y 296.921,Z 463.916,A -85,B 0,C 180,E1 -16287.287,E2 -16287.287} C_VEL
LIN {X 0,Y 297.09,Z 464.866,A -85,B 0,C 180,E1 -16288.644,E2 -16288.644} C_VEL
LIN {X 0,Y 297.1,Z 465.393,A -85,B 0,C 180,E1 -16290,E2 -16290} C_VEL
LIN {X 0,Y 297.043,Z 465.504,A -85,B 0,C 180,E1 -16291.356,E2 -16291.356} C_VEL
LIN {X 0,Y 296.77,Z 464.408,A -85,B 0,C 180,E1 -16294.074,E2 -16294.074} C_VEL
LIN {X 0,Y 296.667,Z 462.962,A -85,B 0,C 180,E1 -16295.744,E2 -16295.744} C_VEL
LIN {X 0,Y 296.857,Z 459.696,A -85,B 0,C 180,E1 -16298.166,E2 -16298.166} C_VEL
LIN {X 0,Y 297.239,Z 455.853,A -85,B 0,C 180,E1 -16300.215,E2 -16300.215} C_VEL
LIN {X 0,Y 297.931,Z 450.915,A -85,B 0,C 180,E1 -16302.258,E2 -16302.258} C_VEL
LIN {X 0,Y 299.313,Z 443.609,A -85,B 0,C 180,E1 -16304.621,E2 -16304.621} C_VEL
LIN {X 0,Y 300.871,Z 435.44,A -85,B 0,C 180,E1 -16306.721,E2 -16306.721} C_VEL
LIN {X 0,Y 302.683,Z 426.197,A -85,B 0,C 180,E1 -16308.618,E2 -16308.618} C_VEL
LIN {X 0,Y 304.758,Z 416.395,A -85,B 0,C 180,E1 -16310.238,E2 -16310.238} C_VEL
LIN {X 0,Y 305.804,Z 409.489,A -85,B 0,C 180,E1 -16311.221,E2 -16311.221} C_VEL
LIN {X 0,Y 306.134,Z 397.441,A -85,B 0,C 180,E1 -16312.766,E2 -16312.766} C_VEL
LIN {X 0,Y 305.346,Z 384.828,A -85,B 0,C 180,E1 -16314.187,E2 -16314.187} C_VEL
LIN {X 0,Y 303.274,Z 371.662,A -85,B 0,C 180,E1 -16315.494,E2 -16315.494} C_VEL
LIN {X 0,Y 299.677,Z 357.425,A -85,B 0,C 180,E1 -16316.793,E2 -16316.793} C_VEL
LIN {X 0,Y 298.782,Z 353.876,A -85,B 0,C 180,E1 -16317.089,E2 -16317.089} C_VEL
LIN {X 0,Y 299.795,Z 347.052,A -85,B 0,C 180,E1 -16321.047,E2 -16321.047} C_VEL
LIN {X 0,Y 301.212,Z 340.185,A -85,B 0,C 180,E1 -16325.25,E2 -16325.25} C_VEL
LIN {X 0,Y 301.834,Z 337.084,A -85,B 0,C 180,E1 -16327.257,E2 -16327.257} C_VEL
LIN {X 0,Y 301.208,Z 332.309,A -85,B 0,C 180,E1 -16330.792,E2 -16330.792} C_VEL
LIN {X 0,Y 300.388,Z 327.771,A -85,B 0,C 180,E1 -16334.58,E2 -16334.58} C_VEL
LIN {X 0,Y 299.612,Z 323.576,A -85,B 0,C 180,E1 -16338.645,E2 -16338.645} C_VEL
LIN {X 0,Y 298.993,Z 320.288,A -85,B 0,C 180,E1 -16342.327,E2 -16342.327} C_VEL
LIN {X 0,Y 298.543,Z 317.887,A -85,B 0,C 180,E1 -16345.599,E2 -16345.599} C_VEL
LIN {X 0,Y 298.401,Z 317.316,A -85,B 0,C 180,E1 -16346.798,E2 -16346.798} C_VEL
LIN {X 0,Y 298.435,Z 317.311,A -85,B 0,C 180,E1 -16350.615,E2 -16350.615} C_VEL
LIN {X 0,Y 298.488,Z 317.305,A -85,B 0,C 180,E1 -16353.474,E2 -16353.474} C_VEL
LIN {X 0,Y 298.44,Z 317.312,A -85,B 0,C 180,E1 -16356.697,E2 -16356.697} C_VEL
LIN {X 0,Y 298.544,Z 317.297,A -85,B 0,C 180,E1 -16360.757,E2 -16360.757} C_VEL
LIN {X 0,Y 298.597,Z 317.288,A -85,B 0,C 180,E1 -16364.995,E2 -16364.995} C_VEL
LIN {X 0,Y 298.587,Z 317.289,A -85,B 0,C 180,E1 -16369.146,E2 -16369.146} C_VEL
LIN {X 0,Y 298.716,Z 317.275,A -85,B 0,C 180,E1 -16371.885,E2 -16371.885} C_VEL
LIN {X 0,Y 298.646,Z 317.286,A -85,B 0,C 180,E1 -16374.598,E2 -16374.598} C_VEL
LIN {X 0,Y 298.926,Z 317.249,A -85,B 0,C 180,E1 -16378.653,E2 -16378.653} C_VEL
LIN {X 0,Y 298.927,Z 317.251,A -85,B 0,C 180,E1 -16381.347,E2 -16381.347} C_VEL
LIN {X 0,Y 298.841,Z 317.262,A -85,B 0,C 180,E1 -16382.696,E2 -16382.696} C_VEL
LIN {X 0,Y 299.022,Z 319.17,A -85,B 0,C 180,E1 -16386.749,E2 -16386.749} C_VEL
LIN {X 0,Y 298.968,Z 320.711,A -85,B 0,C 180,E1 -16389.471,E2 -16389.471} C_VEL
LIN {X 0,Y 298.881,Z 321.827,A -85,B 0,C 180,E1 -16391.1,E2 -16391.1} C_VEL
LIN {X 0,Y 300.214,Z 325.008,A -85,B 0,C 180,E1 -16391.455,E2 -16391.455} C_VEL
LIN {X 0,Y 304.568,Z 334.633,A -85,B 0,C 180,E1 -16392.663,E2 -16392.663} C_VEL
LIN {X 0,Y 308.257,Z 345.409,A -85,B 0,C 180,E1 -16394.018,E2 -16394.018} C_VEL
LIN {X 0,Y 310.611,Z 354.956,A -85,B 0,C 180,E1 -16395.292,E2 -16395.292} C_VEL
LIN {X 0,Y 310.869,Z 357.572,A -85,B 0,C 180,E1 -16395.625,E2 -16395.625} C_VEL
LIN {X 0,Y 309.06,Z 368.677,A -85,B 0,C 180,E1 -16396.933,E2 -16396.933} C_VEL
LIN {X 0,Y 307.164,Z 379.336,A -85,B 0,C 180,E1 -16398.51,E2 -16398.51} C_VEL
LIN {X 0,Y 305.287,Z 388.502,A -85,B 0,C 180,E1 -16400.201,E2 -16400.201} C_VEL
LIN {X 0,Y 303.419,Z 396.792,A -85,B 0,C 180,E1 -16402.102,E2 -16402.102} C_VEL
LIN {X 0,Y 301.699,Z 404.273,A -85,B 0,C 180,E1 -16404.263,E2 -16404.263} C_VEL
LIN {X 0,Y 300.273,Z 410.021,A -85,B 0,C 180,E1 -16406.404,E2 -16406.404} C_VEL
LIN {X 0,Y 299.093,Z 414.751,A -85,B 0,C 180,E1 -16408.74,E2 -16408.74} C_VEL
LIN {X 0,Y 298.093,Z 418.335,A -85,B 0,C 180,E1 -16411.244,E2 -16411.244} C_VEL
LIN {X 0,Y 297.593,Z 419.858,A -85,B 0,C 180,E1 -16412.9,E2 -16412.9} C_VEL
LIN {X 0,Y 297.226,Z 420.824,A -85,B 0,C 180,E1 -16414.575,E2 -16414.575} C_VEL
LIN {X 0,Y 296.953,Z 421.14,A -85,B 0,C 180,E1 -16416.42,E2 -16416.42} C_VEL
LIN {X 0,Y 296.831,Z 420.576,A -85,B 0,C 180,E1 -16418.617,E2 -16418.617} C_VEL
LIN {X 0,Y 296.938,Z 419.004,A -85,B 0,C 180,E1 -16420.765,E2 -16420.765} C_VEL
LIN {X 0,Y 297.323,Z 415.853,A -85,B 0,C 180,E1 -16423.274,E2 -16423.274} C_VEL
LIN {X 0,Y 297.724,Z 412.628,A -85,B 0,C 180,E1 -16425.086,E2 -16425.086} C_VEL
LIN {X 0,Y 298.351,Z 407.208,A -85,B 0,C 180,E1 -16427.403,E2 -16427.403} C_VEL
LIN {X 0,Y 299.221,Z 400.007,A -85,B 0,C 180,E1 -16429.76,E2 -16429.76} C_VEL
LIN {X 0,Y 300.338,Z 391.688,A -85,B 0,C 180,E1 -16431.889,E2 -16431.889} C_VEL
LIN {X 0,Y 301.515,Z 382.667,A -85,B 0,C 180,E1 -16433.739,E2 -16433.739} C_VEL
LIN {X 0,Y 302.731,Z 373.112,A -85,B 0,C 180,E1 -16435.335,E2 -16435.335} C_VEL
LIN {X 0,Y 303.958,Z 362.435,A -85,B 0,C 180,E1 -16436.777,E2 -16436.777} C_VEL
LIN {X 0,Y 305.044,Z 351.101,A -85,B 0,C 180,E1 -16438.001,E2 -16438.001} C_VEL
LIN {X 0,Y 305.229,Z 348.779,A -85,B 0,C 180,E1 -16438.224,E2 -16438.224} C_VEL
LIN {X 0,Y 302.983,Z 337.462,A -85,B 0,C 180,E1 -16439.315,E2 -16439.315} C_VEL
LIN {X 0,Y 299.685,Z 324.216,A -85,B 0,C 180,E1 -16440.351,E2 -16440.351} C_VEL
LIN {X 0,Y 297.707,Z 317.401,A -85,B 0,C 180,E1 -16440.816,E2 -16440.816} C_VEL
LIN {X 0,Y 298.16,Z 317.345,A -85,B 0,C 180,E1 -16444.894,E2 -16444.894} C_VEL
LIN {X 0,Y 298.342,Z 317.321,A -85,B 0,C 180,E1 -16447.857,E2 -16447.857} C_VEL
LIN {X 0,Y 298.464,Z 317.307,A -85,B 0,C 180,E1 -16450.752,E2 -16450.752} C_VEL
LIN {X 0,Y 298.586,Z 317.294,A -85,B 0,C 180,E1 -16454.994,E2 -16454.994} C_VEL
LIN {X 0,Y 298.592,Z 317.293,A -85,B 0,C 180,E1 -16459.146,E2 -16459.146} C_VEL
LIN {X 0,Y 298.703,Z 317.275,A -85,B 0,C 180,E1 -16461.884,E2 -16461.884} C_VEL
LIN {X 0,Y 298.644,Z 317.284,A -85,B 0,C 180,E1 -16464.599,E2 -16464.599} C_VEL
LIN {X 0,Y 298.924,Z 317.251,A -85,B 0,C 180,E1 -16468.653,E2 -16468.653} C_VEL
LIN {X 0,Y 298.923,Z 317.247,A -85,B 0,C 180,E1 -16471.347,E2 -16471.347} C_VEL
LIN {X 0,Y 298.644,Z 317.282,A -85,B 0,C 180,E1 -16475.401,E2 -16475.401} C_VEL
LIN {X 0,Y 298.71,Z 317.277,A -85,B 0,C 180,E1 -16478.822,E2 -16478.822} C_VEL
LIN {X 0,Y 298.554,Z 317.296,A -85,B 0,C 180,E1 -16482.232,E2 -16482.232} C_VEL
LIN {X 0,Y 298.606,Z 317.286,A -85,B 0,C 180,E1 -16485.209,E2 -16485.209} C_VEL
LIN {X 0,Y 298.54,Z 317.295,A -85,B 0,C 180,E1 -16489.243,E2 -16489.243} C_VEL
LIN {X 0,Y 298.458,Z 317.305,A -85,B 0,C 180,E1 -16493.598,E2 -16493.598} C_VEL
LIN {X 0,Y 298.49,Z 317.303,A -85,B 0,C 180,E1 -16496.575,E2 -16496.575} C_VEL
LIN {X 0,Y 298.422,Z 317.31,A -85,B 0,C 180,E1 -16499.641,E2 -16499.641} C_VEL
LIN {X 0,Y 298.397,Z 317.313,A -85,B 0,C 180,E1 -16502.8,E2 -16502.8} C_VEL
LIN {X 0,Y 298.452,Z 317.306,A -85,B 0,C 180,E1 -16506.809,E2 -16506.809} C_VEL
LIN {X 0,Y 298.41,Z 317.312,A -85,B 0,C 180,E1 -16509.486,E2 -16509.486} C_VEL
LIN {X 0,Y 298.4,Z 317.313,A -85,B 0,C 180,E1 -16513.104,E2 -16513.104} C_VEL
LIN {X 0,Y 298.404,Z 317.311,A -85,B 0,C 180,E1 -16516.921,E2 -16516.921} C_VEL
LIN {X 0,Y 298.417,Z 317.311,A -85,B 0,C 180,E1 -16521.004,E2 -16521.004} C_VEL
LIN {X 0,Y 298.42,Z 317.312,A -85,B 0,C 180,E1 -16523.931,E2 -16523.931} C_VEL
LIN {X 0,Y 298.398,Z 317.314,A -85,B 0,C 180,E1 -16527.984,E2 -16527.984} C_VEL
LIN {X 0,Y 298.472,Z 317.304,A -85,B 0,C 180,E1 -16531.905,E2 -16531.905} C_VEL
LIN {X 0,Y 298.487,Z 317.302,A -85,B 0,C 180,E1 -16534.924,E2 -16534.924} C_VEL
LIN {X 0,Y 298.432,Z 317.313,A -85,B 0,C 180,E1 -16539.314,E2 -16539.314} C_VEL
LIN {X 0,Y 298.506,Z 317.298,A -85,B 0,C 180,E1 -16542.178,E2 -16542.178} C_VEL
LIN {X 0,Y 298.588,Z 317.292,A -85,B 0,C 180,E1 -16544.995,E2 -16544.995} C_VEL
LIN {X 0,Y 298.587,Z 317.293,A -85,B 0,C 180,E1 -16549.147,E2 -16549.147} C_VEL
LIN {X 0,Y 298.722,Z 317.272,A -85,B 0,C 180,E1 -16551.885,E2 -16551.885} C_VEL
LIN {X 0,Y 298.656,Z 317.282,A -85,B 0,C 180,E1 -16554.599,E2 -16554.599} C_VEL
LIN {X 0,Y 298.595,Z 317.286,A -85,B 0,C 180,E1 -16555.54,E2 -16555.54} C_VEL
LIN {X 0,Y 297.972,Z 317.368,A -85,B 0,C 180,E1 -16556.667,E2 -16556.667} C_VEL
LIN {X 0,Y 295.322,Z 317.7,A -85,B 0,C 180,E1 -16558.51,E2 -16558.51} C_VEL
LIN {X 0,Y 292.235,Z 318.084,A -85,B 0,C 180,E1 -16560.769,E2 -16560.769} C_VEL
LIN {X 0,Y 291.867,Z 318.126,A -85,B 0,C 180,E1 -16561.547,E2 -16561.547} C_VEL
LIN {X 0,Y 291.696,Z 318.151,A -85,B 0,C 180,E1 -16566.919,E2 -16566.919} C_VEL
LIN {X 0,Y 291.572,Z 318.163,A -85,B 0,C 180,E1 -16569.714,E2 -16569.714} C_VEL
LIN {X 0,Y 291.519,Z 318.169,A -85,B 0,C 180,E1 -16573.951,E2 -16573.951} C_VEL
LIN {X 0,Y 291.443,Z 318.182,A -85,B 0,C 180,E1 -16578.27,E2 -16578.27} C_VEL
LIN {X 0,Y 291.362,Z 318.188,A -85,B 0,C 180,E1 -16581.212,E2 -16581.212} C_VEL
LIN {X 0,Y 291.37,Z 318.19,A -85,B 0,C 180,E1 -16584.208,E2 -16584.208} C_VEL
LIN {X 0,Y 291.365,Z 318.185,A -85,B 0,C 180,E1 -16587.278,E2 -16587.278} C_VEL
LIN {X 0,Y 291.325,Z 318.197,A -85,B 0,C 180,E1 -16590.439,E2 -16590.439} C_VEL
LIN {X 0,Y 291.347,Z 318.193,A -85,B 0,C 180,E1 -16593.698,E2 -16593.698} C_VEL
